# B&R Automation Studio project TD52 (part 82)

#### GridStat.c
```c
/********************************************************************
 * COPYRIGHT -- B&R Industrial Automation GmbH
 ********************************************************************
 * Program: GridStat
 * File: GridStat.c
 * Author: 105055527
 * Last modified by: cadm_kafkama00
 * Created: Mon Sep 05 18:14:57 2016
 * Last modified: Tue Nov 26 15:54:38 2024
 * Model Version: 2.02
 * Description: Detection Algorithm for grid connection.

   HISTORY:
   V1.00  24.07.2020 Keller   created
   V1.01  07.08.2020 Huber  included function block from simulation
   V1.02  29.04.2021 Denk   VectorShift and LVRT function added
   V1.03  31.01.2022 Keller  add input for GCB_On

   V2.00  10.08.2023 Walch  Revision of parametrization, sensitivity and FRT selectivity
   V2.01  22.11.2023 Walch  Include grid observer
   10.01.2024 Walch  Include TP LVRT hold time for weak LVRT blocking
   V2.02  25.11.2024 Walch  Update grid observer for SS mains parallel vs. island plausibility check
 * modified Comment:
 ********************************************************************
 * Implementation of program GridStat
 ********************************************************************
 * Generated with B&R Automation Studio Target for Simulink V6.7.1
 * (ERT based)
 ********************************************************************/

#include "GridStat.h"
#include "GridStat_private.h"

/*  Defines */

/*  Data Types */

/**************************** GLOBAL DATA *************************************/
/*  Definitions */

/*  Declarations  */

/* Forward declaration for local functions */
static real32_T GridStat_mean(const real32_T x[5], struct fGridStat* inst);

/***************************** FILE SCOPE DATA ********************************/

/*************************** FUNCTIONS ****************************************/
int32_T div_nde_s32_floor(int32_T numerator, int32_T denominator, struct fGridStat* inst)
{
  return (((numerator < 0) != (denominator < 0)) && (numerator % denominator !=
           0) ? -1 : 0) + numerator / denominator;
}

/*
 * System initialize for atomic system:
 *    '<S4>/TofLvrtWeakBlk1'
 *    '<S2>/TofMcbFb'
 *    '<S2>/TofReset'
 *    '<S8>/TofAfterFRT'
 *    '<S8>/TofLvrtWeakBlk2'
 */
void GridStat_TofLvrtWeakBlk1_Init(rtDW_TofLvrtWeakBlk1_GridStat *localDW, struct fGridStat* inst)
{
  /* InitializeConditions for DiscreteIntegrator: '<S12>/Discrete-Time Integrator' */
  localDW->DiscreteTimeIntegrator_PrevRese = 2;
  localDW->DiscreteTimeIntegrator_IC_LOADI = 1U;
}

/*
 * Output and update for atomic system:
 *    '<S4>/TofLvrtWeakBlk1'
 *    '<S2>/TofMcbFb'
 *    '<S2>/TofReset'
 *    '<S8>/TofAfterFRT'
 *    '<S8>/TofLvrtWeakBlk2'
 */
void GridStat_TofLvrtWeakBlk1(boolean_T rtu_IN, real32_T rtu_PT,
  rtB_TofLvrtWeakBlk1_GridStat *localB, rtDW_TofLvrtWeakBlk1_GridStat *localDW, struct fGridStat* inst)
{
  real32_T rtb_Switch_l;

  /* Switch: '<S12>/Switch' incorporates:
   *  Constant: '<S12>/Constant1'
   */
  if (rtu_IN) {
    rtb_Switch_l = 0.0F;
  } else {
    rtb_Switch_l = rtu_PT;
  }

  /* End of Switch: '<S12>/Switch' */

  /* DiscreteIntegrator: '<S12>/Discrete-Time Integrator' */
  if (localDW->DiscreteTimeIntegrator_IC_LOADI != 0) {
    localDW->DiscreteTimeIntegrator_DSTATE = rtb_Switch_l;
  }

  if (rtu_IN && (localDW->DiscreteTimeIntegrator_PrevRese <= 0)) {
    localDW->DiscreteTimeIntegrator_DSTATE = rtb_Switch_l;
  }

  /* Logic: '<S12>/Logical Operator1' incorporates:
   *  DiscreteIntegrator: '<S12>/Discrete-Time Integrator'
   *  RelationalOperator: '<S12>/Relational Operator'
   */
  localB->LogicalOperator1 = (localDW->DiscreteTimeIntegrator_DSTATE < rtu_PT);

  /* Update for DiscreteIntegrator: '<S12>/Discrete-Time Integrator' incorporates:
   *  DataTypeConversion: '<S20>/Conversion'
   *  Logic: '<S12>/Logical Operator5'
   */
  localDW->DiscreteTimeIntegrator_IC_LOADI = 0U;
  localDW->DiscreteTimeIntegrator_DSTATE += 0.01F * (real32_T)!rtu_IN;
  localDW->DiscreteTimeIntegrator_PrevRese = (int8_T)rtu_IN;
}

/*
 * System initialize for atomic system:
 *    '<S4>/TpDetNabsProtTrigger'
 *    '<S4>/TpLvrtBlockHold1'
 *    '<S4>/TpLvrtTrigHold1'
 *    '<S4>/TpNabsTrigger'
 *    '<S4>/TpProtTrigger'
 *    '<S8>/TP_PU_trigger'
 *    '<S8>/TpDetVPNTrigger'
 *    '<S8>/TpLvrtBlockHold2'
 *    '<S8>/TpLvrtTrigHold2'
 *    '<S8>/TpNTrigger'
 *    ...
 */
void GridS_TpDetNabsProtTrigger_Init(rtDW_TpDetNabsProtTrigger_GridS *localDW, struct fGridStat* inst)
{
  /* InitializeConditions for UnitDelay: '<S13>/Unit Delay2' */
  localDW->UnitDelay2_DSTATE = true;
}

/*
 * Output and update for atomic system:
 *    '<S4>/TpDetNabsProtTrigger'
 *    '<S4>/TpLvrtBlockHold1'
 *    '<S4>/TpLvrtTrigHold1'
 *    '<S4>/TpNabsTrigger'
 *    '<S4>/TpProtTrigger'
 *    '<S8>/TP_PU_trigger'
 *    '<S8>/TpDetVPNTrigger'
 *    '<S8>/TpLvrtBlockHold2'
 *    '<S8>/TpLvrtTrigHold2'
 *    '<S8>/TpNTrigger'
 *    ...
 */
void GridStat_TpDetNabsProtTrigger(boolean_T rtu_IN, real32_T rtu_PT,
  rtB_TpDetNabsProtTrigger_GridSt *localB, rtDW_TpDetNabsProtTrigger_GridS
  *localDW, struct fGridStat* inst)
{
  real32_T rtb_Switch2;
  real32_T rtb_UkYk1;

  /* Product: '<S24>/delta rise limit' incorporates:
   *  SampleTimeMath: '<S24>/sample time'
   *
   * About '<S24>/sample time':
   *  y = K where K = ( w * Ts )
   */
  rtb_Switch2 = 0.01F;

  /* Outputs for Enabled SubSystem: '<S13>/Enabled Subsystem' incorporates:
   *  EnablePort: '<S22>/Enable'
   */
  /* Logic: '<S13>/Logical Operator3' incorporates:
   *  Logic: '<S13>/Logical Operator2'
   *  UnitDelay: '<S13>/Unit Delay2'
   */
  if ((!rtu_IN) && localDW->UnitDelay2_DSTATE) {
    /* Merge: '<S13>/Merge' incorporates:
     *  Constant: '<S13>/Constant10'
     *  Inport: '<S22>/In1'
     */
    localB->Merge = 0.0F;
  }

  /* End of Logic: '<S13>/Logical Operator3' */
  /* End of Outputs for SubSystem: '<S13>/Enabled Subsystem' */

  /* Outputs for Enabled SubSystem: '<S13>/Enabled Subsystem1' incorporates:
   *  EnablePort: '<S23>/Enable'
   */
  if (rtu_IN) {
    /* Merge: '<S13>/Merge' incorporates:
     *  Inport: '<S23>/In1'
     */
    localB->Merge = rtu_PT;
  }

  /* End of Outputs for SubSystem: '<S13>/Enabled Subsystem1' */

  /* Sum: '<S24>/Difference Inputs1' incorporates:
   *  UnitDelay: '<S24>/Delay Input2'
   */
  rtb_UkYk1 = localB->Merge - localDW->DelayInput2_DSTATE;

  /* Switch: '<S25>/Switch2' incorporates:
   *  RelationalOperator: '<S25>/LowerRelop1'
   */
  if (rtb_UkYk1 <= 0.01F) {
    /* Product: '<S24>/delta fall limit' incorporates:
     *  Constant: '<S13>/Constant9'
     *  SampleTimeMath: '<S24>/sample time'
     *
     * About '<S24>/sample time':
     *  y = K where K = ( w * Ts )
     */
    rtb_Switch2 = -99.99F;

    /* Switch: '<S25>/Switch' incorporates:
     *  RelationalOperator: '<S25>/UpperRelop'
     */
    if (rtb_UkYk1 >= -99.99F) {
      rtb_Switch2 = rtb_UkYk1;
    }

    /* End of Switch: '<S25>/Switch' */
  }

  /* End of Switch: '<S25>/Switch2' */

  /* Sum: '<S24>/Difference Inputs2' incorporates:
   *  UnitDelay: '<S24>/Delay Input2'
   */
  rtb_UkYk1 = rtb_Switch2 + localDW->DelayInput2_DSTATE;

  /* Logic: '<S13>/Logical Operator1' incorporates:
   *  Constant: '<S21>/Constant'
   *  RelationalOperator: '<S13>/Relational Operator1'
   *  RelationalOperator: '<S21>/Compare'
   */
  localB->LogicalOperator1 = ((rtb_UkYk1 > 0.0F) && (rtb_UkYk1 < rtu_PT));

  /* Update for UnitDelay: '<S13>/Unit Delay2' incorporates:
   *  RelationalOperator: '<S13>/Relational Operator3'
   */
  localDW->UnitDelay2_DSTATE = (rtb_UkYk1 >= rtu_PT);

  /* Update for UnitDelay: '<S24>/Delay Input2' */
  localDW->DelayInput2_DSTATE = rtb_UkYk1;
}

/* Function for MATLAB Function: '<S5>/Grid Observer' */
static real32_T GridStat_mean(const real32_T x[5], struct fGridStat* inst)
{
  return ((((x[0] + x[1]) + x[2]) + x[3]) + x[4]) / 5.0F;
}

/* Model step function */
void GridStat_step(RT_MODEL_GridStat *const GridStat_M, struct fGridStat* inst)
{
  struct BlockIO_GridStat *GridStat_B = GridStat_M->blockIO;
  struct D_Work_GridStat *GridStat_DWork = GridStat_M->dwork;
  struct PrevZCSigStates_GridStat *GridStat_PrevZCSigState = GridStat_M->prevZCSigState;
  ExternalOutputs_GridStat *GridStat_Y = (ExternalOutputs_GridStat *)
    GridStat_M->outputs;
  real_T rtb_Switch;
  real_T u0;
  int32_T i;
  int32_T tmp;
  real32_T rtb_Divide4_h;
  real32_T rtb_Product5;
  real32_T rtb_Product6;
  real32_T rtb_Product6_c;
  real32_T rtb_Saturation;
  int16_T rtb_Saturation2;
  int16_T tmp_0;
  boolean_T rtb_AND;
  boolean_T rtb_LogicalOperator3;
  boolean_T rtb_LogicalOperator_b;
  boolean_T rtb_LogicalOperator_i;
  boolean_T rtb_RelationalOperator;
  boolean_T rtb_RelationalOperator3;
  boolean_T rtb_RelationalOperator3_dy;
  boolean_T rtb_RelationalOperator_b;
  boolean_T rtb_Switch6;
  boolean_T rtb_trigger_LVRT_l;
  boolean_T rtb_trigger_N;
  boolean_T rtb_trigger_P;
  boolean_T rtb_trigger_PU;
  boolean_T rtb_trigger_U;

  /* S-Function (bur_bus_in): '<Root>/Bus Input' */
  GridStat_B->BusInput = inst->Para;

  /* S-Function (bur_bus_in): '<Root>/Bus Input2' */
  GridStat_B->BusInput2 = inst->In;

  /* Logic: '<S2>/AND' */
  rtb_AND = (GridStat_B->BusInput2.bGCB_On && GridStat_B->BusInput2.bMCB_On);

  /* Outputs for Atomic SubSystem: '<S2>/TofMcbFb' */
  GridStat_TofLvrtWeakBlk1(rtb_AND, GridStat_B->BusInput.rTi_Tof_MCBfb,
    &GridStat_B->TofMcbFb, &GridStat_DWork->TofMcbFb, inst);

  /* End of Outputs for SubSystem: '<S2>/TofMcbFb' */

  /* Saturate: '<S4>/Saturation5' */
  if (GridStat_B->BusInput.rN_Nom >= 1.0F) {
    rtb_Saturation = GridStat_B->BusInput.rN_Nom;
  } else {
    rtb_Saturation = 1.0F;
  }

  /* End of Saturate: '<S4>/Saturation5' */

  /* RelationalOperator: '<S4>/Relational Operator' incorporates:
   *  Abs: '<S4>/Abs'
   *  Abs: '<S4>/Abs1'
   *  Product: '<S4>/Product4'
   *  Sum: '<S4>/Sum'
   */
  rtb_RelationalOperator = ((real32_T)fabs(GridStat_B->BusInput2.rN_engAct -
    rtb_Saturation) > (real32_T)fabs(rtb_Saturation *
    GridStat_B->BusInput.rThrs_DeltaN_norm));

  /* Outputs for Atomic SubSystem: '<S4>/TpNabsTrigger' */
  /* SignalConversion generated from: '<S4>/Bus Selector2' */
  GridStat_TpDetNabsProtTrigger(rtb_RelationalOperator,
    GridStat_B->BusInput.rTi_Tp_DetectActive, &GridStat_B->TpNabsTrigger,
    &GridStat_DWork->TpNabsTrigger, inst);

  /* End of Outputs for SubSystem: '<S4>/TpNabsTrigger' */

  /* Gain: '<S4>/rpm2omega' */
  rtb_Saturation = 0.104719758F * GridStat_B->BusInput2.rN_engAct;

  /* Outputs for Atomic SubSystem: '<S4>/Speed_filter' */
  /* Logic: '<S11>/Logical Operator' incorporates:
   *  Constant: '<S11>/Constant'
   *  Logic: '<S11>/Logical Operator1'
   *  RelationalOperator: '<S11>/Relational Operator'
   */
  rtb_LogicalOperator_i = (GridStat_B->BusInput2.bReset ||
    (GridStat_B->BusInput.rTi_Filt_speed <= 0.0F));

  /* DiscreteIntegrator: '<S11>/Discrete-Time Integrator' */
  if (GridStat_DWork->DiscreteTimeIntegrator_IC_LOADI != 0) {
    GridStat_DWork->DiscreteTimeIntegrator_DSTATE_j = rtb_Saturation;
  }

  if (rtb_LogicalOperator_i || (GridStat_DWork->DiscreteTimeIntegrator_PrevRese
       != 0)) {
    GridStat_DWork->DiscreteTimeIntegrator_DSTATE_j = rtb_Saturation;
  }

  /* Switch: '<S18>/Switch' incorporates:
   *  Abs: '<S18>/Abs'
   *  RelationalOperator: '<S18>/Relational Operator'
   */
  if (2.22044605E-16F >= (real32_T)fabs(GridStat_B->BusInput.rTi_Filt_speed)) {
    rtb_Product5 = 2.22044605E-16F;
  } else {
    rtb_Product5 = GridStat_B->BusInput.rTi_Filt_speed;
  }

  /* End of Switch: '<S18>/Switch' */

  /* Product: '<S11>/Divide4' incorporates:
   *  DiscreteIntegrator: '<S11>/Discrete-Time Integrator'
   *  Sum: '<S11>/Sum4'
   */
  rtb_Divide4_h = (rtb_Saturation -
                   GridStat_DWork->DiscreteTimeIntegrator_DSTATE_j) /
    rtb_Product5;

  /* Update for DiscreteIntegrator: '<S11>/Discrete-Time Integrator' */
  GridStat_DWork->DiscreteTimeIntegrator_IC_LOADI = 0U;
  GridStat_DWork->DiscreteTimeIntegrator_DSTATE_j += 0.01F * rtb_Divide4_h;
  GridStat_DWork->DiscreteTimeIntegrator_PrevRese = (int8_T)
    rtb_LogicalOperator_i;

  /* End of Outputs for SubSystem: '<S4>/Speed_filter' */

  /* Gain: '<S4>/W2kW' */
  rtb_Product6 = 1000.0F * GridStat_B->BusInput.rP_Nom;

  /* Outputs for Atomic SubSystem: '<S4>/Speed_filter' */
  /* Switch: '<S11>/Switch1' incorporates:
   *  Constant: '<S11>/Constant'
   */
  if (rtb_LogicalOperator_i) {
    rtb_Divide4_h = 0.0F;
  }

  /* End of Switch: '<S11>/Switch1' */
  /* End of Outputs for SubSystem: '<S4>/Speed_filter' */

  /* Saturate: '<S4>/Saturation' */
  if (rtb_Product6 < 1.0F) {
    rtb_Product6 = 1.0F;
  }

  /* End of Saturate: '<S4>/Saturation' */

  /* Product: '<S4>/Product2' incorporates:
   *  Product: '<S4>/Product1'
   */
  rtb_Saturation = rtb_Saturation * rtb_Divide4_h *
    GridStat_B->BusInput.rJ_Engine / rtb_Product6;

  /* RelationalOperator: '<S4>/Relational Operator2' */
  rtb_LogicalOperator_i = (rtb_Saturation >
    GridStat_B->BusInput.rProt_Norm_limit);

  /* Outputs for Atomic SubSystem: '<S4>/TpProtTrigger' */
  /* SignalConversion generated from: '<S4>/Bus Selector2' */
  GridStat_TpDetNabsProtTrigger(rtb_LogicalOperator_i,
    GridStat_B->BusInput.rTi_Tp_DetectActive, &GridStat_B->TpProtTrigger,
    &GridStat_DWork->TpProtTrigger, inst);

  /* End of Outputs for SubSystem: '<S4>/TpProtTrigger' */

  /* RelationalOperator: '<S4>/Relational Operator3' */
  rtb_RelationalOperator3 = (GridStat_B->BusInput2.rU_norm <=
    GridStat_B->BusInput.rThrs_LVRT_norm);

  /* Saturate: '<S4>/Saturation1' */
  if (GridStat_B->BusInput.rTi_sampleRate >= 0.001F) {
    /* Saturate: '<S8>/Saturation' incorporates:
     *  Saturate: '<S8>/Saturation1'
     */
    rtb_Divide4_h = GridStat_B->BusInput.rTi_sampleRate;
  } else {
    /* Saturate: '<S8>/Saturation' incorporates:
     *  Saturate: '<S8>/Saturation1'
     */
    rtb_Divide4_h = 0.001F;
  }

  /* Saturate: '<S4>/Saturation4' incorporates:
   *  DataTypeConversion: '<S4>/Cast1'
   */
  if (GridStat_B->BusInput.iSamples_Tp_LVRT_hold > 10000.0F) {
    rtb_Product5 = 10000.0F;
  } else if (GridStat_B->BusInput.iSamples_Tp_LVRT_hold < 1.0F) {
    rtb_Product5 = 1.0F;
  } else {
    rtb_Product5 = GridStat_B->BusInput.iSamples_Tp_LVRT_hold;
  }

  /* End of Saturate: '<S4>/Saturation4' */

  /* Product: '<S4>/Product6' incorporates:
   *  Saturate: '<S4>/Saturation1'
   */
  rtb_Product6 = rtb_Divide4_h * rtb_Product5;

  /* Outputs for Atomic SubSystem: '<S4>/TpLvrtBlockHold1' */
  /* Logic: '<S4>/Logical Operator2' */
  GridStat_TpDetNabsProtTrigger((rtb_RelationalOperator3 ||
    GridStat_B->BusInput2.bLVRT), rtb_Product6, &GridStat_B->TpLvrtBlockHold1,
    &GridStat_DWork->TpLvrtBlockHold1, inst);

  /* End of Outputs for SubSystem: '<S4>/TpLvrtBlockHold1' */

  /* Saturate: '<S4>/Saturation2' incorporates:
   *  Constant: '<S4>/Constant1'
   *  DataTypeConversion: '<S4>/Cast'
   *  Sum: '<S4>/Sum3'
   */
  if (10.0F - (real32_T)GridStat_B->BusInput.iSensitivity_WeakBlocking > 10.0F)
  {
    rtb_Product5 = 10.0F;
  } else if (10.0F - (real32_T)GridStat_B->BusInput.iSensitivity_WeakBlocking <
             1.0F) {
    rtb_Product5 = 1.0F;
  } else {
    rtb_Product5 = 10.0F - (real32_T)
      GridStat_B->BusInput.iSensitivity_WeakBlocking;
  }

  /* End of Saturate: '<S4>/Saturation2' */

  /* Outputs for Atomic SubSystem: '<S4>/TofLvrtWeakBlk1' */
  /* Product: '<S4>/Product7' incorporates:
   *  Saturate: '<S4>/Saturation1'
   */
  GridStat_TofLvrtWeakBlk1(rtb_RelationalOperator3, rtb_Product5 * rtb_Divide4_h,
    &GridStat_B->TofLvrtWeakBlk1, &GridStat_DWork->TofLvrtWeakBlk1, inst);

  /* End of Outputs for SubSystem: '<S4>/TofLvrtWeakBlk1' */

  /* Outputs for Atomic SubSystem: '<S4>/TpLvrtTrigHold1' */
  GridStat_TpDetNabsProtTrigger(GridStat_B->BusInput2.bLVRT, rtb_Product6,
    &GridStat_B->TpLvrtTrigHold1, &GridStat_DWork->TpLvrtTrigHold1, inst);

  /* End of Outputs for SubSystem: '<S4>/TpLvrtTrigHold1' */

  /* Switch: '<S4>/Switch1' incorporates:
   *  Constant: '<S4>/Constant'
   *  Logic: '<S4>/Logical Operator1'
   *  Logic: '<S4>/Logical Operator11'
   *  Logic: '<S4>/Logical Operator3'
   *  Logic: '<S4>/NOT2'
   *  Switch: '<S4>/Switch5'
   */
  if (rtb_RelationalOperator && (GridStat_B->BusInput.bN_BypassFRTBlocking &&
       GridStat_B->BusInput.bN_BypassFRTBlocking_speedAbs)) {
    rtb_RelationalOperator3 = false;
  } else if ((!GridStat_B->BusInput.bWeakFRTBlocking) ||
             (!GridStat_B->BusInput.bWeakFRTBlocking_speedAbs)) {
    /* Switch: '<S4>/Switch5' */
    rtb_RelationalOperator3 = GridStat_B->TpLvrtBlockHold1.LogicalOperator1;
  } else {
    /* Switch: '<S4>/Switch5' incorporates:
     *  Logic: '<S4>/Logical Operator9'
     */
    rtb_RelationalOperator3 = (GridStat_B->TofLvrtWeakBlk1.LogicalOperator1 &&
      GridStat_B->TpLvrtTrigHold1.LogicalOperator1);
  }

  /* End of Switch: '<S4>/Switch1' */

  /* Logic: '<S4>/NOT' */
  rtb_Switch6 = !rtb_RelationalOperator3;

  /* Switch: '<S4>/Switch4' incorporates:
   *  Saturate: '<S4>/Saturation1'
   */
  if (rtb_Switch6) {
    rtb_Product6 = GridStat_B->BusInput.rTi_Tp_DetectActive;
  } else {
    rtb_Product6 = rtb_Divide4_h;
  }

  /* End of Switch: '<S4>/Switch4' */

  /* Outputs for Atomic SubSystem: '<S4>/TpDetNabsProtTrigger' */
  /* Logic: '<S4>/Logical Operator4' incorporates:
   *  Logic: '<S4>/Logical Operator'
   */
  GridStat_TpDetNabsProtTrigger(((GridStat_B->TpNabsTrigger.LogicalOperator1 ||
    GridStat_B->TpProtTrigger.LogicalOperator1) && rtb_Switch6), rtb_Product6,
    &GridStat_B->TpDetNabsProtTrigger, &GridStat_DWork->TpDetNabsProtTrigger, inst);

  /* End of Outputs for SubSystem: '<S4>/TpDetNabsProtTrigger' */

  /* Saturate: '<S8>/Saturation2' */
  if (GridStat_B->BusInput.iSamples_derivative_PU > 10) {
    rtb_Saturation2 = 10;
  } else if (GridStat_B->BusInput.iSamples_derivative_PU < 1) {
    rtb_Saturation2 = 1;
  } else {
    rtb_Saturation2 = GridStat_B->BusInput.iSamples_derivative_PU;
  }

  /* End of Saturate: '<S8>/Saturation2' */

  /* Product: '<S8>/Product' */
  rtb_Product6 = (real32_T)rtb_Saturation2 * rtb_Divide4_h;

  /* RelationalOperator: '<S8>/Relational Operator3' */
  rtb_RelationalOperator3_dy = (GridStat_B->BusInput2.rU_norm <=
    GridStat_B->BusInput.rThrs_LVRT_norm);

  /* Saturate: '<S8>/Saturation7' incorporates:
   *  Constant: '<S8>/Constant1'
   *  DataTypeConversion: '<S8>/Cast'
   *  Sum: '<S8>/Sum3'
   */
  if (10.0F - (real32_T)GridStat_B->BusInput.iSensitivity_WeakBlocking > 10.0F)
  {
    rtb_Product5 = 10.0F;
  } else if (10.0F - (real32_T)GridStat_B->BusInput.iSensitivity_WeakBlocking <
             1.0F) {
    rtb_Product5 = 1.0F;
  } else {
    rtb_Product5 = 10.0F - (real32_T)
      GridStat_B->BusInput.iSensitivity_WeakBlocking;
  }

  /* End of Saturate: '<S8>/Saturation7' */

  /* Outputs for Atomic SubSystem: '<S8>/TofLvrtWeakBlk2' */
  /* Product: '<S8>/Product7' */
  GridStat_TofLvrtWeakBlk1(rtb_RelationalOperator3_dy, rtb_Product5 *
    rtb_Divide4_h, &GridStat_B->TofLvrtWeakBlk2,
    &GridStat_DWork->TofLvrtWeakBlk2, inst);

  /* End of Outputs for SubSystem: '<S8>/TofLvrtWeakBlk2' */

  /* Saturate: '<S8>/Saturation4' */
  if (GridStat_B->BusInput.iSamples_Tp_LVRT_hold > 10000) {
    tmp_0 = 10000;
  } else if (GridStat_B->BusInput.iSamples_Tp_LVRT_hold < 1) {
    tmp_0 = 1;
  } else {
    tmp_0 = GridStat_B->BusInput.iSamples_Tp_LVRT_hold;
  }

  /* End of Saturate: '<S8>/Saturation4' */

  /* Product: '<S8>/Product6' */
  rtb_Product6_c = rtb_Divide4_h * (real32_T)tmp_0;

  /* Outputs for Atomic SubSystem: '<S8>/TpLvrtTrigHold2' */
  GridStat_TpDetNabsProtTrigger(GridStat_B->BusInput2.bLVRT, rtb_Product6_c,
    &GridStat_B->TpLvrtTrigHold2, &GridStat_DWork->TpLvrtTrigHold2, inst);

  /* End of Outputs for SubSystem: '<S8>/TpLvrtTrigHold2' */

  /* Logic: '<S8>/Logical Operator9' */
  rtb_trigger_LVRT_l = (GridStat_B->TofLvrtWeakBlk2.LogicalOperator1 &&
                        GridStat_B->TpLvrtTrigHold2.LogicalOperator1);

  /* Saturate: '<S8>/Saturation6' */
  if (GridStat_B->BusInput.iSamples_Tof_U_norm_FRTBlock > 1000) {
    tmp_0 = 1000;
  } else if (GridStat_B->BusInput.iSamples_Tof_U_norm_FRTBlock < 1) {
    tmp_0 = 1;
  } else {
    tmp_0 = GridStat_B->BusInput.iSamples_Tof_U_norm_FRTBlock;
  }

  /* End of Saturate: '<S8>/Saturation6' */

  /* Outputs for Atomic SubSystem: '<S8>/TofAfterFRT' */
  /* Product: '<S8>/Product8' */
  GridStat_TofLvrtWeakBlk1(rtb_trigger_LVRT_l, (real32_T)tmp_0 * rtb_Divide4_h,
    &GridStat_B->TofAfterFRT, &GridStat_DWork->TofAfterFRT, inst);

  /* End of Outputs for SubSystem: '<S8>/TofAfterFRT' */

  /* Switch: '<S8>/Switch7' incorporates:
   *  Logic: '<S8>/NOT3'
   */
  if (!GridStat_B->TofAfterFRT.LogicalOperator1) {
    rtb_Product5 = GridStat_B->BusInput.rThrs_U_norm;
  } else {
    rtb_Product5 = GridStat_B->BusInput.rThrs_U_norm_FRTBlock;
  }

  /* End of Switch: '<S8>/Switch7' */

  /* RelationalOperator: '<S8>/Relational Operator' incorporates:
   *  Abs: '<S8>/Abs'
   *  Product: '<S8>/Product1'
   *  S-Function (sfix_udelay): '<S8>/Tapped Delay'
   *  Selector: '<S8>/Selector'
   *  Sum: '<S8>/Sum'
   */
  rtb_trigger_U = ((real32_T)fabs(GridStat_DWork->TappedDelay_X[rtb_Saturation2
    - 1] - GridStat_B->BusInput2.rU_norm) / rtb_Product6 >= rtb_Product5);

  /* Saturate: '<S8>/Saturation3' */
  if (GridStat_B->BusInput.iSamples_Tp_detect_VPN > 1000) {
    tmp_0 = 1000;
  } else if (GridStat_B->BusInput.iSamples_Tp_detect_VPN < 1) {
    tmp_0 = 1;
  } else {
    tmp_0 = GridStat_B->BusInput.iSamples_Tp_detect_VPN;
  }

  /* End of Saturate: '<S8>/Saturation3' */

  /* Product: '<S8>/Product5' */
  rtb_Product5 = (real32_T)tmp_0 * rtb_Divide4_h;

  /* Outputs for Atomic SubSystem: '<S8>/TpUTrigger' */
  GridStat_TpDetNabsProtTrigger(rtb_trigger_U, rtb_Product5,
    &GridStat_B->TpUTrigger, &GridStat_DWork->TpUTrigger, inst);

  /* End of Outputs for SubSystem: '<S8>/TpUTrigger' */

  /* RelationalOperator: '<S8>/Relational Operator1' incorporates:
   *  Abs: '<S8>/Abs1'
   *  Product: '<S8>/Product2'
   *  S-Function (sfix_udelay): '<S8>/Tapped Delay1'
   *  Selector: '<S8>/Selector'
   *  Selector: '<S8>/Selector1'
   *  Sum: '<S8>/Sum1'
   */
  rtb_trigger_P = ((real32_T)fabs(GridStat_DWork->TappedDelay1_X[rtb_Saturation2
    - 1] - GridStat_B->BusInput2.rP_norm) / rtb_Product6 >=
                   GridStat_B->BusInput.rThrs_P_norm);

  /* Outputs for Atomic SubSystem: '<S8>/TpPTrigger' */
  GridStat_TpDetNabsProtTrigger(rtb_trigger_P, rtb_Product5,
    &GridStat_B->TpPTrigger, &GridStat_DWork->TpPTrigger, inst);

  /* End of Outputs for SubSystem: '<S8>/TpPTrigger' */

  /* Switch: '<S8>/Switch1' incorporates:
   *  Logic: '<S8>/Logical Operator5'
   *  Logic: '<S8>/Logical Operator6'
   *  Switch: '<S8>/Switch'
   */
  if (GridStat_B->BusInput.bLimitedTriggerTime) {
    rtb_RelationalOperator_b = GridStat_B->TpUTrigger.LogicalOperator1;
    rtb_LogicalOperator3 = GridStat_B->TpPTrigger.LogicalOperator1;
  } else {
    rtb_RelationalOperator_b = (GridStat_B->TpUTrigger.LogicalOperator1 ||
      rtb_trigger_U);
    rtb_LogicalOperator3 = (GridStat_B->TpPTrigger.LogicalOperator1 ||
      rtb_trigger_P);
  }

  /* End of Switch: '<S8>/Switch1' */

  /* Logic: '<S8>/Logical Operator' */
  rtb_trigger_PU = (rtb_RelationalOperator_b && rtb_LogicalOperator3);

  /* Outputs for Atomic SubSystem: '<S8>/TP_PU_trigger' */
  GridStat_TpDetNabsProtTrigger(rtb_trigger_PU, rtb_Product5,
    &GridStat_B->TP_PU_trigger, &GridStat_DWork->TP_PU_trigger, inst);

  /* End of Outputs for SubSystem: '<S8>/TP_PU_trigger' */

  /* Saturate: '<S8>/Saturation5' */
  if (GridStat_B->BusInput.iSamples_derivative_N > 10) {
    rtb_Saturation2 = 10;
  } else if (GridStat_B->BusInput.iSamples_derivative_N < 1) {
    rtb_Saturation2 = 1;
  } else {
    rtb_Saturation2 = GridStat_B->BusInput.iSamples_derivative_N;
  }

  /* End of Saturate: '<S8>/Saturation5' */

  /* RelationalOperator: '<S8>/Relational Operator2' incorporates:
   *  Abs: '<S8>/Abs2'
   *  Product: '<S8>/Product3'
   *  Product: '<S8>/Product4'
   *  S-Function (sfix_udelay): '<S8>/Tapped Delay2'
   *  Selector: '<S8>/Selector2'
   *  Sum: '<S8>/Sum2'
   */
  rtb_trigger_N = (GridStat_B->BusInput.rThrs_N_eng <= 1.0F / (rtb_Divide4_h *
    (real32_T)rtb_Saturation2) * (real32_T)fabs(GridStat_DWork->
    TappedDelay2_X[rtb_Saturation2 - 1] - GridStat_B->BusInput2.rN_engAct));

  /* Outputs for Atomic SubSystem: '<S8>/TpNTrigger' */
  GridStat_TpDetNabsProtTrigger(rtb_trigger_N, rtb_Product5,
    &GridStat_B->TpNTrigger, &GridStat_DWork->TpNTrigger, inst);

  /* End of Outputs for SubSystem: '<S8>/TpNTrigger' */

  /* Outputs for Atomic SubSystem: '<S8>/TpLvrtBlockHold2' */
  /* Logic: '<S8>/Logical Operator2' */
  GridStat_TpDetNabsProtTrigger((rtb_RelationalOperator3_dy ||
    GridStat_B->BusInput2.bLVRT), rtb_Product6_c, &GridStat_B->TpLvrtBlockHold2,
    &GridStat_DWork->TpLvrtBlockHold2, inst);

  /* End of Outputs for SubSystem: '<S8>/TpLvrtBlockHold2' */

  /* Switch: '<S8>/Switch6' incorporates:
   *  Constant: '<S8>/Constant'
   *  Logic: '<S8>/Logical Operator10'
   *  Logic: '<S8>/Logical Operator11'
   *  Logic: '<S8>/Logical Operator12'
   *  Logic: '<S8>/NOT2'
   *  Switch: '<S8>/Switch5'
   */
  if (rtb_RelationalOperator && (GridStat_B->BusInput.bN_BypassFRTBlocking &&
       GridStat_B->BusInput.bN_BypassFRTBlocking_VPN)) {
    rtb_Switch6 = false;
  } else if ((!GridStat_B->BusInput.bWeakFRTBlocking) ||
             (!GridStat_B->BusInput.bWeakFRTBlocking_VPN)) {
    /* Switch: '<S8>/Switch5' */
    rtb_Switch6 = GridStat_B->TpLvrtBlockHold2.LogicalOperator1;
  } else {
    rtb_Switch6 = rtb_trigger_LVRT_l;
  }

  /* End of Switch: '<S8>/Switch6' */

  /* Logic: '<S8>/NOT' */
  rtb_trigger_LVRT_l = !rtb_Switch6;

  /* Switch: '<S8>/Switch2' incorporates:
   *  Logic: '<S8>/Logical Operator7'
   */
  if (GridStat_B->BusInput.bLimitedTriggerTime) {
    rtb_RelationalOperator_b = GridStat_B->TP_PU_trigger.LogicalOperator1;
  } else {
    rtb_RelationalOperator_b = (GridStat_B->TP_PU_trigger.LogicalOperator1 ||
      rtb_trigger_PU);
  }

  /* End of Switch: '<S8>/Switch2' */

  /* Switch: '<S8>/Switch3' incorporates:
   *  Logic: '<S8>/Logical Operator8'
   *  Logic: '<S8>/NOT1'
   */
  if (!GridStat_B->BusInput.bLimitedTriggerTime) {
    rtb_LogicalOperator3 = (rtb_trigger_N ||
      GridStat_B->TpNTrigger.LogicalOperator1);
  } else {
    rtb_LogicalOperator3 = GridStat_B->TpNTrigger.LogicalOperator1;
  }

  /* End of Switch: '<S8>/Switch3' */

  /* Switch: '<S8>/Switch4' */
  if (rtb_trigger_LVRT_l) {
    rtb_Divide4_h = GridStat_B->BusInput.rTi_Tp_DetectActive;
  }

  /* End of Switch: '<S8>/Switch4' */

  /* Outputs for Atomic SubSystem: '<S8>/TpDetVPNTrigger' */
  /* Logic: '<S8>/Logical Operator4' incorporates:
   *  Logic: '<S8>/Logical Operator1'
   *  Logic: '<S8>/Logical Operator3'
   */
  GridStat_TpDetNabsProtTrigger((((rtb_RelationalOperator_b &&
    rtb_LogicalOperator3) || GridStat_B->BusInput2.bVectorShift) &&
    rtb_trigger_LVRT_l), rtb_Divide4_h, &GridStat_B->TpDetVPNTrigger,
    &GridStat_DWork->TpDetVPNTrigger, inst);

  /* End of Outputs for SubSystem: '<S8>/TpDetVPNTrigger' */

  /* MATLAB Function: '<S5>/Grid Observer' */
  /* MATLAB Function 'detection + correction: transition to Island/Smooth Detection/Grid Observer': '<S52>:1' */
  /* '<S52>:1:2' */
  tmp = 10 - GridStat_B->BusInput.iSensitivity_SmoothDetection;
  if (10 - GridStat_B->BusInput.iSensitivity_SmoothDetection > 32767) {
    tmp = 32767;
  }

  if ((!GridStat_DWork->U_past_not_empty) || GridStat_B->BusInput2.bReset) {
    GridStat_DWork->ctr_U = 0;
    for (i = 0; i < 1000; i++) {
      GridStat_DWork->U_past[i] = GridStat_B->BusInput2.rU_norm;
    }

    GridStat_DWork->U_past_not_empty = true;
  }

  i = GridStat_DWork->ctr_U + 1;
  if (GridStat_DWork->ctr_U + 1 > 32767) {
    i = 32767;
  }

  GridStat_DWork->U_past[i - 1] = GridStat_B->BusInput2.rU_norm;
  rtb_Divide4_h = 0.0F;
  for (rtb_Saturation2 = 0; rtb_Saturation2 < 1000; rtb_Saturation2++) {
    i = GridStat_DWork->ctr_U - rtb_Saturation2;
    if (i < -32768) {
      i = -32768;
    }

    i = (int16_T)((int16_T)i - (int16_T)((int16_T)div_nde_s32_floor((int16_T)i,
      1000, inst) * 1000)) + 1;
    if (i > 32767) {
      i = 32767;
    }

    rtb_Divide4_h += GridStat_DWork->U_past[i - 1];
  }

  rtb_Divide4_h /= 1000.0F;
  i = GridStat_DWork->ctr_U + 1;
  if (GridStat_DWork->ctr_U + 1 > 32767) {
    i = 32767;
  }

  GridStat_DWork->ctr_U = (int16_T)i;
  if (GridStat_DWork->ctr_U >= 1000) {
    GridStat_DWork->ctr_U = 0;
  }

  if ((!GridStat_DWork->err_past_not_empty) || GridStat_B->BusInput2.bReset) {
    GridStat_DWork->ctr_err = 0;
    GridStat_DWork->ctr_acterr = 0;
    GridStat_DWork->ctr_release = 0;
    for (i = 0; i < 1000; i++) {
      GridStat_DWork->err_past[i] = 0.0F;
    }

    GridStat_DWork->err_past_not_empty = true;
    GridStat_DWork->err_min = 1.0E+6F;
    GridStat_DWork->err_act = 0.0F;
    GridStat_DWork->err_max = 0.0F;
    GridStat_DWork->flag_window = true;
    for (i = 0; i < 5; i++) {
      GridStat_DWork->err_act_temp[i] = 0.0F;
    }
  }

  i = GridStat_DWork->ctr_err + 1;
  if (GridStat_DWork->ctr_err + 1 > 32767) {
    i = 32767;
  }

  if (1.0F >= GridStat_B->BusInput.rN_Nom) {
    rtb_Product5 = 1.0F;
  } else {
    rtb_Product5 = GridStat_B->BusInput.rN_Nom;
  }

  GridStat_DWork->err_past[i - 1] = (real32_T)fabs
    (GridStat_B->BusInput2.rN_engAct / rtb_Product5 - 1.0F);
  rtb_Product6 = GridStat_DWork->err_past[0];
  for (i = 0; i < 999; i++) {
    rtb_Product6 += GridStat_DWork->err_past[i + 1];
  }

  rtb_trigger_LVRT_l = true;
  if (GridStat_DWork->ctr_release < 6000) {
    i = GridStat_DWork->ctr_release + 1;
    if (GridStat_DWork->ctr_release + 1 > 32767) {
      i = 32767;
    }

    GridStat_DWork->ctr_release = (int16_T)i;
    rtb_trigger_LVRT_l = false;
  }

  if (GridStat_DWork->flag_window && rtb_trigger_LVRT_l) {
    i = GridStat_DWork->ctr_acterr + 1;
    if (GridStat_DWork->ctr_acterr + 1 > 32767) {
      i = 32767;
    }

    GridStat_DWork->err_act_temp[i - 1] = rtb_Product6 / 1000.0F;
    i = GridStat_DWork->ctr_acterr + 1;
    if (GridStat_DWork->ctr_acterr + 1 > 32767) {
      i = 32767;
    }

    GridStat_DWork->ctr_acterr = (int16_T)i;
    GridStat_DWork->flag_window = false;
  }

  rtb_Product6 = GridStat_DWork->err_act_temp[0];
  rtb_Product6_c = GridStat_mean(GridStat_DWork->err_act_temp, inst);
  rtb_Product5 = GridStat_DWork->err_act_temp[0];
  if (GridStat_DWork->err_act_temp[0] < GridStat_DWork->err_act_temp[1]) {
    rtb_Product6 = GridStat_DWork->err_act_temp[1];
  }

  if (GridStat_DWork->err_act_temp[0] > GridStat_DWork->err_act_temp[1]) {
    rtb_Product5 = GridStat_DWork->err_act_temp[1];
  }

  if (rtb_Product6 < GridStat_DWork->err_act_temp[2]) {
    rtb_Product6 = GridStat_DWork->err_act_temp[2];
  }

  if (rtb_Product5 > GridStat_DWork->err_act_temp[2]) {
    rtb_Product5 = GridStat_DWork->err_act_temp[2];
  }

  if (rtb_Product6 < GridStat_DWork->err_act_temp[3]) {
    rtb_Product6 = GridStat_DWork->err_act_temp[3];
  }

  if (rtb_Product5 > GridStat_DWork->err_act_temp[3]) {
    rtb_Product5 = GridStat_DWork->err_act_temp[3];
  }

  if (rtb_Product6 < GridStat_DWork->err_act_temp[4]) {
    rtb_Product6 = GridStat_DWork->err_act_temp[4];
  }

  if (rtb_Product5 > GridStat_DWork->err_act_temp[4]) {
    rtb_Product5 = GridStat_DWork->err_act_temp[4];
  }

  if (((real32_T)fabs(rtb_Product6 - rtb_Product6_c) < rtb_Product6_c) &&
      ((real32_T)fabs(rtb_Product6_c - rtb_Product5) < rtb_Product6_c)) {
    GridStat_DWork->err_act = GridStat_mean(GridStat_DWork->err_act_temp, inst);
  }

  if ((GridStat_DWork->err_act < GridStat_DWork->err_min) &&
      (GridStat_DWork->err_act > 1.0E-8F)) {
    GridStat_DWork->err_min = GridStat_DWork->err_act;
  }

  if (GridStat_DWork->err_act > GridStat_DWork->err_max) {
    GridStat_DWork->err_max = GridStat_DWork->err_act;
  }

  if (GridStat_DWork->ctr_acterr > 4) {
    GridStat_DWork->ctr_acterr = 0;
  }

  i = GridStat_DWork->ctr_err + 1;
  if (GridStat_DWork->ctr_err + 1 > 32767) {
    i = 32767;
  }

  GridStat_DWork->ctr_err = (int16_T)i;
  if (GridStat_DWork->ctr_err >= 1000) {
    GridStat_DWork->ctr_err = 0;
    GridStat_DWork->flag_window = true;
  }

  if ((!GridStat_DWork->err_past_Q_not_empty) || GridStat_B->BusInput2.bReset) {
    GridStat_DWork->ctr_err_Q = 0;
    GridStat_DWork->ctr_acterr_Q = 0;
    GridStat_DWork->ctr_release_Q = 0;
    for (i = 0; i < 1000; i++) {
      GridStat_DWork->err_past_Q[i] = 0.0F;
    }

    GridStat_DWork->err_past_Q_not_empty = true;
    GridStat_DWork->err_min_Q = 1.0E+6F;
    GridStat_DWork->err_act_Q = 0.0F;
    GridStat_DWork->err_max_Q = 0.0F;
    GridStat_DWork->flag_window_Q = true;
    for (i = 0; i < 5; i++) {
      GridStat_DWork->err_act_temp_Q[i] = 0.0F;
    }
  }

  i = GridStat_DWork->ctr_err_Q + 1;
  if (GridStat_DWork->ctr_err_Q + 1 > 32767) {
    i = 32767;
  }

  GridStat_DWork->err_past_Q[i - 1] = (real32_T)fabs
    (GridStat_B->BusInput2.rU_norm - rtb_Divide4_h);
  rtb_Divide4_h = GridStat_DWork->err_past_Q[0];
  for (i = 0; i < 999; i++) {
    rtb_Divide4_h += GridStat_DWork->err_past_Q[i + 1];
  }

  rtb_trigger_LVRT_l = true;
  if (GridStat_DWork->ctr_release_Q < 6000) {
    i = GridStat_DWork->ctr_release_Q + 1;
    if (GridStat_DWork->ctr_release_Q + 1 > 32767) {
      i = 32767;
    }

    GridStat_DWork->ctr_release_Q = (int16_T)i;
    rtb_trigger_LVRT_l = false;
  }

  if (GridStat_DWork->flag_window_Q && rtb_trigger_LVRT_l) {
    i = GridStat_DWork->ctr_acterr_Q + 1;
    if (GridStat_DWork->ctr_acterr_Q + 1 > 32767) {
      i = 32767;
    }

    GridStat_DWork->err_act_temp_Q[i - 1] = rtb_Divide4_h / 1000.0F;
    i = GridStat_DWork->ctr_acterr_Q + 1;
    if (GridStat_DWork->ctr_acterr_Q + 1 > 32767) {
      i = 32767;
    }

    GridStat_DWork->ctr_acterr_Q = (int16_T)i;
    GridStat_DWork->flag_window_Q = false;
  }

  rtb_Divide4_h = GridStat_DWork->err_act_temp_Q[0];
  rtb_Product6 = GridStat_mean(GridStat_DWork->err_act_temp_Q, inst);
  rtb_Product6_c = GridStat_DWork->err_act_temp_Q[0];
  if (GridStat_DWork->err_act_temp_Q[0] < GridStat_DWork->err_act_temp_Q[1]) {
    rtb_Divide4_h = GridStat_DWork->err_act_temp_Q[1];
  }

  if (GridStat_DWork->err_act_temp_Q[0] > GridStat_DWork->err_act_temp_Q[1]) {
    rtb_Product6_c = GridStat_DWork->err_act_temp_Q[1];
  }

  if (rtb_Divide4_h < GridStat_DWork->err_act_temp_Q[2]) {
    rtb_Divide4_h = GridStat_DWork->err_act_temp_Q[2];
  }

  if (rtb_Product6_c > GridStat_DWork->err_act_temp_Q[2]) {
    rtb_Product6_c = GridStat_DWork->err_act_temp_Q[2];
  }

  if (rtb_Divide4_h < GridStat_DWork->err_act_temp_Q[3]) {
    rtb_Divide4_h = GridStat_DWork->err_act_temp_Q[3];
  }

  if (rtb_Product6_c > GridStat_DWork->err_act_temp_Q[3]) {
    rtb_Product6_c = GridStat_DWork->err_act_temp_Q[3];
  }

  if (rtb_Divide4_h < GridStat_DWork->err_act_temp_Q[4]) {
    rtb_Divide4_h = GridStat_DWork->err_act_temp_Q[4];
  }

  if (rtb_Product6_c > GridStat_DWork->err_act_temp_Q[4]) {
    rtb_Product6_c = GridStat_DWork->err_act_temp_Q[4];
  }

  if (((real32_T)fabs(rtb_Divide4_h - rtb_Product6) < rtb_Product6) &&
      ((real32_T)fabs(rtb_Product6 - rtb_Product6_c) < rtb_Product6)) {
    GridStat_DWork->err_act_Q = GridStat_mean(GridStat_DWork->err_act_temp_Q, inst);
  }

  if ((GridStat_DWork->err_act_Q < GridStat_DWork->err_min_Q) &&
      (GridStat_DWork->err_act_Q > 1.0E-8F)) {
    GridStat_DWork->err_min_Q = GridStat_DWork->err_act_Q;
  }

  if (GridStat_DWork->err_act_Q > GridStat_DWork->err_max_Q) {
    GridStat_DWork->err_max_Q = GridStat_DWork->err_act_Q;
  }

  if (GridStat_DWork->ctr_acterr_Q > 4) {
    GridStat_DWork->ctr_acterr_Q = 0;
  }

  i = GridStat_DWork->ctr_err_Q + 1;
  if (GridStat_DWork->ctr_err_Q + 1 > 32767) {
    i = 32767;
  }

  GridStat_DWork->ctr_err_Q = (int16_T)i;
  if (GridStat_DWork->ctr_err_Q >= 1000) {
    GridStat_DWork->ctr_err_Q = 0;
    GridStat_DWork->flag_window_Q = true;
  }

  rtb_RelationalOperator_b = false;
  rtb_Divide4_h = (real32_T)(int16_T)tmp / 2.0F;
  if ((int16_T)tmp == 0) {
    rtb_Divide4_h = 0.25F;
  }

  if (1.0E-8F >= GridStat_DWork->err_min) {
    rtb_Product5 = 1.0E-8F;
  } else {
    rtb_Product5 = GridStat_DWork->err_min;
  }

  if (GridStat_DWork->err_act / rtb_Product5 > rtb_Divide4_h * 15.0F) {
    rtb_RelationalOperator_b = true;
  } else {
    if (1.0E-8F >= GridStat_DWork->err_min_Q) {
      rtb_Product5 = 1.0E-8F;
    } else {
      rtb_Product5 = GridStat_DWork->err_min_Q;
    }

    if (GridStat_DWork->err_act_Q / rtb_Product5 > rtb_Divide4_h * 3.5F) {
      rtb_RelationalOperator_b = true;
    }
  }

  /* MultiPortSwitch: '<S2>/Multiport Switch' incorporates:
   *  Logic: '<S2>/Logical Operator'
   *  Logic: '<S2>/Logical Operator1'
   */
  /* '<S52>:1:2' */
  switch (GridStat_B->BusInput.iDetectMode) {
   case 1:
    rtb_trigger_LVRT_l = GridStat_B->TpDetNabsProtTrigger.LogicalOperator1;
    break;

   case 2:
    rtb_trigger_LVRT_l = GridStat_B->TpDetVPNTrigger.LogicalOperator1;
    break;

   default:
    rtb_trigger_LVRT_l = (GridStat_B->TpDetNabsProtTrigger.LogicalOperator1 ||
                          GridStat_B->TpDetVPNTrigger.LogicalOperator1 ||
                          (GridStat_B->BusInput.bEnable_SmoothDetection &&
      rtb_RelationalOperator_b));
    break;
  }

  /* End of MultiPortSwitch: '<S2>/Multiport Switch' */

  /* Logic: '<S2>/Logical Operator3' incorporates:
   *  Logic: '<S2>/Logical Operator5'
   */
  rtb_LogicalOperator3 = ((rtb_AND || GridStat_B->TofMcbFb.LogicalOperator1) &&
    GridStat_B->BusInput.bEnable && rtb_trigger_LVRT_l);

  /* Outputs for Atomic SubSystem: '<S2>/TofReset' */
  GridStat_TofLvrtWeakBlk1(rtb_LogicalOperator3,
    GridStat_B->BusInput.rTi_Filt_factorNoffsetCorr, &GridStat_B->TofReset,
    &GridStat_DWork->TofReset, inst);

  /* End of Outputs for SubSystem: '<S2>/TofReset' */

  /* Outputs for Atomic SubSystem: '<S2>/Filter' */
  /* RelationalOperator: '<S3>/Relational Operator' incorporates:
   *  Constant: '<S3>/Constant'
   */
  rtb_trigger_LVRT_l = (GridStat_B->BusInput.rTi_Filt_factorNoffsetCorr > 0.0F);

  /* Logic: '<S3>/Logical Operator' incorporates:
   *  Logic: '<S3>/Logical Operator1'
   */
  rtb_LogicalOperator_b = (GridStat_B->TofReset.LogicalOperator1 ||
    (!rtb_trigger_LVRT_l));

  /* DiscreteIntegrator: '<S3>/Discrete-Time Integrator' */
  if (rtb_LogicalOperator_b || (GridStat_DWork->DiscreteTimeIntegrator_PrevRe_g
       != 0)) {
    GridStat_DWork->DiscreteTimeIntegrator_DSTATE = 0.0;
  }

  /* Switch: '<S3>/Switch' incorporates:
   *  Constant: '<S2>/Constant12'
   *  DiscreteIntegrator: '<S3>/Discrete-Time Integrator'
   */
  if (rtb_trigger_LVRT_l) {
    rtb_Switch = GridStat_DWork->DiscreteTimeIntegrator_DSTATE;
  } else {
    rtb_Switch = 1.0;
  }

  /* End of Switch: '<S3>/Switch' */

  /* Switch: '<S9>/Switch' incorporates:
   *  Abs: '<S9>/Abs'
   *  RelationalOperator: '<S9>/Relational Operator'
   */
  if (2.22044605E-16F >= (real32_T)fabs
      (GridStat_B->BusInput.rTi_Filt_factorNoffsetCorr)) {
    rtb_Product5 = 2.22044605E-16F;
  } else {
    rtb_Product5 = GridStat_B->BusInput.rTi_Filt_factorNoffsetCorr;
  }

  /* End of Switch: '<S9>/Switch' */

  /* Update for DiscreteIntegrator: '<S3>/Discrete-Time Integrator' incorporates:
   *  Constant: '<S2>/Constant12'
   *  Product: '<S3>/Divide4'
   *  Sum: '<S3>/Sum4'
   */
  GridStat_DWork->DiscreteTimeIntegrator_DSTATE += (1.0 -
    GridStat_DWork->DiscreteTimeIntegrator_DSTATE) / rtb_Product5 * 0.01;
  GridStat_DWork->DiscreteTimeIntegrator_PrevRe_g = (int8_T)
    rtb_LogicalOperator_b;

  /* End of Outputs for SubSystem: '<S2>/Filter' */

  /* Logic: '<S2>/Logical Operator4' */
  rtb_trigger_LVRT_l = !rtb_AND;

  /* Delay: '<S2>/IslandDetected' */
  GridStat_DWork->icLoad = ((((GridStat_PrevZCSigState->IslandDetected_Reset_ZCE
    == 1) != (int32_T)GridStat_B->BusInput2.bReset) &&
    (GridStat_PrevZCSigState->IslandDetected_Reset_ZCE != 3)) ||
    GridStat_B->BusInput2.bReset || GridStat_DWork->icLoad);
  GridStat_PrevZCSigState->IslandDetected_Reset_ZCE =
    GridStat_B->BusInput2.bReset;
  GridStat_DWork->IslandDetected_DSTATE = ((!GridStat_DWork->icLoad) &&
    GridStat_DWork->IslandDetected_DSTATE);

  /* Switch: '<S2>/Switch1' incorporates:
   *  Delay: '<S2>/IslandDetected'
   *  Logic: '<S2>/Logical Operator6'
   */
  if (rtb_trigger_LVRT_l || rtb_LogicalOperator3) {
    rtb_AND = rtb_LogicalOperator3;
  } else {
    rtb_AND = GridStat_DWork->IslandDetected_DSTATE;
  }

  /* End of Switch: '<S2>/Switch1' */

  /* Logic: '<Root>/Logical Operator' incorporates:
   *  Logic: '<S2>/Logical Operator2'
   */
  GridStat_Y->Out.bGridStatus = ((!rtb_trigger_LVRT_l) && (!rtb_AND));

  /* Product: '<S2>/Product' */
  u0 = rtb_Switch * GridStat_B->BusInput2.rN_F_Offset_Norm;

  /* MinMax: '<S2>/MinMax1' */
  if (u0 <= GridStat_B->BusInput2.rN_F_Offset_Norm) {
    /* BusCreator: '<Root>/Bus Creator1' incorporates:
     *  DataTypeConversion: '<Root>/Data Type Conversion1'
     *  Outport: '<Root>/Out'
     */
    GridStat_Y->Out.rN_F_Offset_Norm_corr = (real32_T)u0;
  } else {
    /* BusCreator: '<Root>/Bus Creator1' incorporates:
     *  Outport: '<Root>/Out'
     */
    GridStat_Y->Out.rN_F_Offset_Norm_corr =
      GridStat_B->BusInput2.rN_F_Offset_Norm;
  }

  /* End of MinMax: '<S2>/MinMax1' */

  /* BusCreator generated from: '<Root>/dbg' incorporates:
   *  DataTypeConversion: '<S2>/Data Type Conversion1'
   *  MATLAB Function: '<S5>/Grid Observer'
   *  Outport: '<Root>/dbg'
   */
  GridStat_Y->dbg.rProt_norm = rtb_Saturation;
  GridStat_Y->dbg.bDetSpeedRise =
    GridStat_B->TpDetNabsProtTrigger.LogicalOperator1;
  GridStat_Y->dbg.bDetIslandVPN = GridStat_B->TpDetVPNTrigger.LogicalOperator1;
  GridStat_Y->dbg.trigger_Nabs = rtb_RelationalOperator;
  GridStat_Y->dbg.trigger_Prot = rtb_LogicalOperator_i;
  GridStat_Y->dbg.trigger_PU = rtb_trigger_PU;
  GridStat_Y->dbg.trigger_N = rtb_trigger_N;
  GridStat_Y->dbg.trigger_U = rtb_trigger_U;
  GridStat_Y->dbg.trigger_P = rtb_trigger_P;
  GridStat_Y->dbg.trigger_VS = GridStat_B->BusInput2.bVectorShift;
  GridStat_Y->dbg.block_LVRT_VPN = rtb_Switch6;
  GridStat_Y->dbg.trigger_LVRT_NoDelay = rtb_RelationalOperator3_dy;
  GridStat_Y->dbg.rCorrFac_rN_set_Norm = (real32_T)rtb_Switch;
  GridStat_Y->dbg.block_LVRT_speedAbs = rtb_RelationalOperator3;
  GridStat_Y->dbg.bDetGridObserver = rtb_RelationalOperator_b;
  for (i = 0; i < 9; i++) {
    GridStat_Y->dbg.ru_obs[i] = 0.0F;
    GridStat_Y->dbg.ru_obs_strong[i] = 0.0F;
    GridStat_Y->dbg.ru_obs3[i] = 0.0F;
  }

  GridStat_Y->dbg.ry_obs[0] = 0.0F;
  GridStat_Y->dbg.ry_obs[1] = 0.0F;
  for (i = 0; i < 5; i++) {
    GridStat_Y->dbg.rx_obs[i] = 0.0F;
    GridStat_Y->dbg.rx_obs_strong[i] = 0.0F;
    GridStat_Y->dbg.rx_obs3[i] = 0.0F;
    GridStat_Y->dbg.rcorr[i] = 0.0F;
    GridStat_Y->dbg.rcorr_strong[i] = 0.0F;
    GridStat_Y->dbg.rcorr3[i] = 0.0F;
  }

  /* End of BusCreator generated from: '<Root>/dbg' */

  /* S-Function (bur_bus_out): '<Root>/Bus Output' incorporates:
   *  Outport: '<Root>/Out'
   */
  inst->Out = GridStat_Y->Out;

  /* BusCreator generated from: '<Root>/Bus Output1' incorporates:
   *  DataTypeConversion: '<S2>/Data Type Conversion1'
   *  MATLAB Function: '<S5>/Grid Observer'
   */
  GridStat_B->BusConversion_InsertedFor_BusOu.rProt_norm = rtb_Saturation;
  GridStat_B->BusConversion_InsertedFor_BusOu.bDetSpeedRise =
    GridStat_B->TpDetNabsProtTrigger.LogicalOperator1;
  GridStat_B->BusConversion_InsertedFor_BusOu.bDetIslandVPN =
    GridStat_B->TpDetVPNTrigger.LogicalOperator1;
  GridStat_B->BusConversion_InsertedFor_BusOu.trigger_Nabs =
    rtb_RelationalOperator;
  GridStat_B->BusConversion_InsertedFor_BusOu.trigger_Prot =
    rtb_LogicalOperator_i;
  GridStat_B->BusConversion_InsertedFor_BusOu.trigger_PU = rtb_trigger_PU;
  GridStat_B->BusConversion_InsertedFor_BusOu.trigger_N = rtb_trigger_N;
  GridStat_B->BusConversion_InsertedFor_BusOu.trigger_U = rtb_trigger_U;
  GridStat_B->BusConversion_InsertedFor_BusOu.trigger_P = rtb_trigger_P;
  GridStat_B->BusConversion_InsertedFor_BusOu.trigger_VS =
    GridStat_B->BusInput2.bVectorShift;
  GridStat_B->BusConversion_InsertedFor_BusOu.block_LVRT_VPN = rtb_Switch6;
  GridStat_B->BusConversion_InsertedFor_BusOu.trigger_LVRT_NoDelay =
    rtb_RelationalOperator3_dy;
  GridStat_B->BusConversion_InsertedFor_BusOu.rCorrFac_rN_set_Norm = (real32_T)
    rtb_Switch;
  GridStat_B->BusConversion_InsertedFor_BusOu.block_LVRT_speedAbs =
    rtb_RelationalOperator3;
  GridStat_B->BusConversion_InsertedFor_BusOu.bDetGridObserver =
    rtb_RelationalOperator_b;
  for (i = 0; i < 9; i++) {
    GridStat_B->BusConversion_InsertedFor_BusOu.ru_obs[i] = 0.0F;
    GridStat_B->BusConversion_InsertedFor_BusOu.ru_obs_strong[i] = 0.0F;
    GridStat_B->BusConversion_InsertedFor_BusOu.ru_obs3[i] = 0.0F;
  }

  GridStat_B->BusConversion_InsertedFor_BusOu.ry_obs[0] = 0.0F;
  GridStat_B->BusConversion_InsertedFor_BusOu.ry_obs[1] = 0.0F;
  for (i = 0; i < 5; i++) {
    GridStat_B->BusConversion_InsertedFor_BusOu.rx_obs[i] = 0.0F;
    GridStat_B->BusConversion_InsertedFor_BusOu.rx_obs_strong[i] = 0.0F;
    GridStat_B->BusConversion_InsertedFor_BusOu.rx_obs3[i] = 0.0F;
    GridStat_B->BusConversion_InsertedFor_BusOu.rcorr[i] = 0.0F;
    GridStat_B->BusConversion_InsertedFor_BusOu.rcorr_strong[i] = 0.0F;
    GridStat_B->BusConversion_InsertedFor_BusOu.rcorr3[i] = 0.0F;
  }

  /* End of BusCreator generated from: '<Root>/Bus Output1' */

  /* S-Function (bur_bus_out): '<Root>/Bus Output1' */
  inst->Dbg = GridStat_B->BusConversion_InsertedFor_BusOu;

  /* S-Function (bur_bus_in): '<Root>/Bus Input1' */
  GridStat_B->BusInput1 = inst->Perm;

  /* UnitDelay: '<S1>/Unit Delay' */
  GridStat_B->UnitDelay = GridStat_DWork->UnitDelay_DSTATE;

  /* S-Function (bur_out): '<Root>/Bus Output2' */
  inst->Version = GridStat_B->UnitDelay;
  for (i = 0; i < 9; i++) {
    /* Update for S-Function (sfix_udelay): '<S8>/Tapped Delay' */
    GridStat_DWork->TappedDelay_X[9 - i] = GridStat_DWork->TappedDelay_X[8 - i];

    /* Update for S-Function (sfix_udelay): '<S8>/Tapped Delay1' */
    GridStat_DWork->TappedDelay1_X[9 - i] = GridStat_DWork->TappedDelay1_X[8 - i];

    /* Update for S-Function (sfix_udelay): '<S8>/Tapped Delay2' */
    GridStat_DWork->TappedDelay2_X[9 - i] = GridStat_DWork->TappedDelay2_X[8 - i];

    /* Update for S-Function (sfix_udelay): '<S5>/Tapped Delay' */
    GridStat_DWork->TappedDelay_X_l[9 - i] = GridStat_DWork->TappedDelay_X_l[8 -
      i];

    /* Update for S-Function (sfix_udelay): '<S5>/Tapped Delay2' */
    GridStat_DWork->TappedDelay2_X_b[9 - i] = GridStat_DWork->TappedDelay2_X_b[8
      - i];

    /* Update for S-Function (sfix_udelay): '<S5>/Tapped Delay3' */
    GridStat_DWork->TappedDelay3_X[9 - i] = GridStat_DWork->TappedDelay3_X[8 - i];

    /* Update for S-Function (sfix_udelay): '<S5>/Tapped Delay5' */
    GridStat_DWork->TappedDelay5_X[9 - i] = GridStat_DWork->TappedDelay5_X[8 - i];

    /* Update for S-Function (sfix_udelay): '<S5>/Tapped Delay4' */
    GridStat_DWork->TappedDelay4_X[9 - i] = GridStat_DWork->TappedDelay4_X[8 - i];

    /* Update for S-Function (sfix_udelay): '<S5>/Tapped Delay1' */
    GridStat_DWork->TappedDelay1_X_m[9 - i] = GridStat_DWork->TappedDelay1_X_m[8
      - i];
  }

  /* Update for S-Function (sfix_udelay): '<S8>/Tapped Delay' */
  GridStat_DWork->TappedDelay_X[0] = GridStat_B->BusInput2.rU_norm;

  /* Update for S-Function (sfix_udelay): '<S8>/Tapped Delay1' */
  GridStat_DWork->TappedDelay1_X[0] = GridStat_B->BusInput2.rP_norm;

  /* Update for S-Function (sfix_udelay): '<S8>/Tapped Delay2' */
  GridStat_DWork->TappedDelay2_X[0] = GridStat_B->BusInput2.rN_engAct;

  /* Update for S-Function (sfix_udelay): '<S5>/Tapped Delay' */
  GridStat_DWork->TappedDelay_X_l[0] = GridStat_B->BusInput2.rp2s_norm;

  /* Update for S-Function (sfix_udelay): '<S5>/Tapped Delay2' */
  GridStat_DWork->TappedDelay2_X_b[0] = GridStat_B->BusInput2.rP_norm;

  /* Update for S-Function (sfix_udelay): '<S5>/Tapped Delay3' */
  GridStat_DWork->TappedDelay3_X[0] = GridStat_B->BusInput2.rN_engAct;

  /* Update for S-Function (sfix_udelay): '<S5>/Tapped Delay5' */
  GridStat_DWork->TappedDelay5_X[0] = GridStat_B->BusInput2.rQ_norm;

  /* Update for S-Function (sfix_udelay): '<S5>/Tapped Delay4' */
  GridStat_DWork->TappedDelay4_X[0] = GridStat_B->BusInput2.rU_norm;

  /* Update for S-Function (sfix_udelay): '<S5>/Tapped Delay1' */
  GridStat_DWork->TappedDelay1_X_m[0] = GridStat_B->BusInput2.rUexc_norm;

  /* Update for Delay: '<S2>/IslandDetected' */
  GridStat_DWork->icLoad = false;
  GridStat_DWork->IslandDetected_DSTATE = rtb_AND;

  /* Update for UnitDelay: '<S1>/Unit Delay' */
  GridStat_DWork->UnitDelay_DSTATE = 202U;
}

/* Model initialize function */
void GridStat_initialize(RT_MODEL_GridStat *const GridStat_M, struct fGridStat* inst)
{
  struct D_Work_GridStat *GridStat_DWork = GridStat_M->dwork;
  struct PrevZCSigStates_GridStat *GridStat_PrevZCSigState = GridStat_M->prevZCSigState;
  GridStat_PrevZCSigState->IslandDetected_Reset_ZCE = UNINITIALIZED_ZCSIG;

  /* InitializeConditions for Delay: '<S2>/IslandDetected' */
  GridStat_DWork->icLoad = true;

  /* SystemInitialize for Atomic SubSystem: '<S2>/TofMcbFb' */
  GridStat_TofLvrtWeakBlk1_Init(&GridStat_DWork->TofMcbFb, inst);

  /* End of SystemInitialize for SubSystem: '<S2>/TofMcbFb' */

  /* SystemInitialize for Atomic SubSystem: '<S4>/TpNabsTrigger' */
  GridS_TpDetNabsProtTrigger_Init(&GridStat_DWork->TpNabsTrigger, inst);

  /* End of SystemInitialize for SubSystem: '<S4>/TpNabsTrigger' */

  /* SystemInitialize for Atomic SubSystem: '<S4>/Speed_filter' */
  /* InitializeConditions for DiscreteIntegrator: '<S11>/Discrete-Time Integrator' */
  GridStat_DWork->DiscreteTimeIntegrator_IC_LOADI = 1U;

  /* End of SystemInitialize for SubSystem: '<S4>/Speed_filter' */

  /* SystemInitialize for Atomic SubSystem: '<S4>/TpProtTrigger' */
  GridS_TpDetNabsProtTrigger_Init(&GridStat_DWork->TpProtTrigger, inst);

  /* End of SystemInitialize for SubSystem: '<S4>/TpProtTrigger' */

  /* SystemInitialize for Atomic SubSystem: '<S4>/TpLvrtBlockHold1' */
  GridS_TpDetNabsProtTrigger_Init(&GridStat_DWork->TpLvrtBlockHold1, inst);

  /* End of SystemInitialize for SubSystem: '<S4>/TpLvrtBlockHold1' */

  /* SystemInitialize for Atomic SubSystem: '<S4>/TofLvrtWeakBlk1' */
  GridStat_TofLvrtWeakBlk1_Init(&GridStat_DWork->TofLvrtWeakBlk1, inst);

  /* End of SystemInitialize for SubSystem: '<S4>/TofLvrtWeakBlk1' */

  /* SystemInitialize for Atomic SubSystem: '<S4>/TpLvrtTrigHold1' */
  GridS_TpDetNabsProtTrigger_Init(&GridStat_DWork->TpLvrtTrigHold1, inst);

  /* End of SystemInitialize for SubSystem: '<S4>/TpLvrtTrigHold1' */

  /* SystemInitialize for Atomic SubSystem: '<S4>/TpDetNabsProtTrigger' */
  GridS_TpDetNabsProtTrigger_Init(&GridStat_DWork->TpDetNabsProtTrigger, inst);

  /* End of SystemInitialize for SubSystem: '<S4>/TpDetNabsProtTrigger' */

  /* SystemInitialize for Atomic SubSystem: '<S8>/TofLvrtWeakBlk2' */
  GridStat_TofLvrtWeakBlk1_Init(&GridStat_DWork->TofLvrtWeakBlk2, inst);

  /* End of SystemInitialize for SubSystem: '<S8>/TofLvrtWeakBlk2' */

  /* SystemInitialize for Atomic SubSystem: '<S8>/TpLvrtTrigHold2' */
  GridS_TpDetNabsProtTrigger_Init(&GridStat_DWork->TpLvrtTrigHold2, inst);

  /* End of SystemInitialize for SubSystem: '<S8>/TpLvrtTrigHold2' */

  /* SystemInitialize for Atomic SubSystem: '<S8>/TofAfterFRT' */
  GridStat_TofLvrtWeakBlk1_Init(&GridStat_DWork->TofAfterFRT, inst);

  /* End of SystemInitialize for SubSystem: '<S8>/TofAfterFRT' */

  /* SystemInitialize for Atomic SubSystem: '<S8>/TpUTrigger' */
  GridS_TpDetNabsProtTrigger_Init(&GridStat_DWork->TpUTrigger, inst);

  /* End of SystemInitialize for SubSystem: '<S8>/TpUTrigger' */

  /* SystemInitialize for Atomic SubSystem: '<S8>/TpPTrigger' */
  GridS_TpDetNabsProtTrigger_Init(&GridStat_DWork->TpPTrigger, inst);

  /* End of SystemInitialize for SubSystem: '<S8>/TpPTrigger' */

  /* SystemInitialize for Atomic SubSystem: '<S8>/TP_PU_trigger' */
  GridS_TpDetNabsProtTrigger_Init(&GridStat_DWork->TP_PU_trigger, inst);

  /* End of SystemInitialize for SubSystem: '<S8>/TP_PU_trigger' */

  /* SystemInitialize for Atomic SubSystem: '<S8>/TpNTrigger' */
  GridS_TpDetNabsProtTrigger_Init(&GridStat_DWork->TpNTrigger, inst);

  /* End of SystemInitialize for SubSystem: '<S8>/TpNTrigger' */

  /* SystemInitialize for Atomic SubSystem: '<S8>/TpLvrtBlockHold2' */
  GridS_TpDetNabsProtTrigger_Init(&GridStat_DWork->TpLvrtBlockHold2, inst);

  /* End of SystemInitialize for SubSystem: '<S8>/TpLvrtBlockHold2' */

  /* SystemInitialize for Atomic SubSystem: '<S8>/TpDetVPNTrigger' */
  GridS_TpDetNabsProtTrigger_Init(&GridStat_DWork->TpDetVPNTrigger, inst);

  /* End of SystemInitialize for SubSystem: '<S8>/TpDetVPNTrigger' */

  /* SystemInitialize for Atomic SubSystem: '<S2>/TofReset' */
  GridStat_TofLvrtWeakBlk1_Init(&GridStat_DWork->TofReset, inst);

  /* End of SystemInitialize for SubSystem: '<S2>/TofReset' */
}

/* Model terminate function */
void GridStat_terminate(RT_MODEL_GridStat *const GridStat_M, struct fGridStat* inst)
{
  /* (no terminate code required) */
  UNUSED_PARAMETER(GridStat_M);
}

/*======================== TOOL VERSION INFORMATION ==========================*
 * MATLAB 9.11 (R2021b)14-May-2021                                            *
 * Simulink 10.4 (R2021b)14-May-2021                                          *
 * Simulink Coder 9.6 (R2021b)14-May-2021                                     *
 * Embedded Coder 7.7 (R2021b)14-May-2021                                     *
 * Stateflow 10.5 (R2021b)14-May-2021                                         *
 *============================================================================*/

/*======================= LICENSE IN USE INFORMATION =========================*
 * matlab                                                                     *
 * matlab_coder                                                               *
 * real-time_workshop                                                         *
 * rtw_embedded_coder                                                         *
 * simulink                                                                   *
 *============================================================================*/
```

#### GridStat.h
```c
/********************************************************************
 * COPYRIGHT -- B&R Industrial Automation GmbH
 ********************************************************************
 * Program: GridStat
 * File: GridStat.h
 * Author: 105055527
 * Last modified by: cadm_kafkama00
 * Created: Mon Sep 05 18:14:57 2016
 * Last modified: Tue Nov 26 15:54:38 2024
 * Model Version: 2.02
 * Description: Detection Algorithm for grid connection.

   HISTORY:
   V1.00  24.07.2020 Keller   created
   V1.01  07.08.2020 Huber  included function block from simulation
   V1.02  29.04.2021 Denk   VectorShift and LVRT function added
   V1.03  31.01.2022 Keller  add input for GCB_On

   V2.00  10.08.2023 Walch  Revision of parametrization, sensitivity and FRT selectivity
   V2.01  22.11.2023 Walch  Include grid observer
   10.01.2024 Walch  Include TP LVRT hold time for weak LVRT blocking
   V2.02  25.11.2024 Walch  Update grid observer for SS mains parallel vs. island plausibility check
 * modified Comment:
 ********************************************************************
 * Header for program GridStat
 ********************************************************************
 * Generated with B&R Automation Studio Target for Simulink V6.7.1
 * (ERT based)
 ********************************************************************/

#ifndef RTW_HEADER_GridStat_h_
#define RTW_HEADER_GridStat_h_
#include <math.h>
#ifndef GridStat_COMMON_INCLUDES_
#define GridStat_COMMON_INCLUDES_
#include "rtwtypes.h"
#include "zero_crossing_types.h"
#endif                                 /* GridStat_COMMON_INCLUDES_ */

#include "GridStat_types.h"
#include "lGridStat.h"
/* Beginning of Dynamic TypeDefs: */
/* End of Dynamic TypeDefs: */
#ifndef MIN
#define MIN(a,b)	((a) < (b) ? (a) : (b))
#endif

#ifndef MAX
#define MAX(a,b)	((a) > (b) ? (a) : (b))
#endif

#ifndef AST_ROUND
#define AST_ROUND(x) ((x)>=0?(long long)((x)+0.5):(long long)((x)-0.5))
#endif

#include "rt_defines.h"

/* Macros for accessing real-time model data structure */
#ifndef rtmGetBlockIO
#define rtmGetBlockIO(rtm)             ((rtm)->blockIO)
#endif

#ifndef rtmSetBlockIO
#define rtmSetBlockIO(rtm, val)        ((rtm)->blockIO = (val))
#endif

#ifndef rtmGetPrevZCSigState
#define rtmGetPrevZCSigState(rtm)      ((rtm)->prevZCSigState)
#endif

#ifndef rtmSetPrevZCSigState
#define rtmSetPrevZCSigState(rtm, val) ((rtm)->prevZCSigState = (val))
#endif

#ifndef rtmGetRootDWork
#define rtmGetRootDWork(rtm)           ((rtm)->dwork)
#endif

#ifndef rtmSetRootDWork
#define rtmSetRootDWork(rtm, val)      ((rtm)->dwork = (val))
#endif

#ifndef rtmGetY
#define rtmGetY(rtm)                   ((rtm)->outputs)
#endif

#ifndef rtmSetY
#define rtmSetY(rtm, val)              ((rtm)->outputs = (val))
#endif

#ifndef rtmGetErrorStatus
#define rtmGetErrorStatus(rtm)         ((rtm)->errorStatus)
#endif

#ifndef rtmSetErrorStatus
#define rtmSetErrorStatus(rtm, val)    ((rtm)->errorStatus = (val))
#endif

#ifndef MIN
#define MIN(a,b)                       ((a) < (b) ? (a) : (b))
#endif

#ifndef MAX
#define MAX(a,b)                       ((a) > (b) ? (a) : (b))
#endif

#ifndef AST_ROUND
#define AST_ROUND(x)                   ((x)>=0?(long long)((x)+0.5):(long long)((x)-0.5))
#endif

/* user code (top of header file) */
/***************************************************************************************************
 * COPYRIGHT -- INNIO Jenbacher GmbH & CO OG
 ****************************************************************************************************
 * Program:            GridStat
 * Author:             cadm_kafkama00
 * Created:            26.11.2024 15:54
 ****************************************************************************************************
 * MODEL INFORMATION
 ****************************************************************************************************
 * Model Name:         C:\Users\kafkama00\Documents\Git\JenCtrLib\Controllers\GridStatusDetection\GridStat.slx
 * Model Version:      2.02
 * Simulink Version:   R2021b
 * B&R Target:         V6.7.1
 * Description:        Detection Algorithm for grid connection.
 *
 *                     HISTORY:
 *                     V1.00  24.07.2020 Keller   created
 *                     V1.01  07.08.2020 Huber  included function block from simulation
 *                     V1.02  29.04.2021 Denk   VectorShift and LVRT function added
 *                     V1.03  31.01.2022 Keller  add input for GCB_On
 *
 *                     V2.00  10.08.2023 Walch  Revision of parametrization, sensitivity and FRT selectivity
 *                     V2.01  22.11.2023 Walch  Include grid observer
 *                                10.01.2024 Walch  Include TP LVRT hold time for weak LVRT blocking
 *                     V2.02  25.11.2024 Walch  Update grid observer for SS mains parallel vs. island plausibility check
 ****************************************************************************************************
 * Last Modified By:   walchin00
 * Last Modified Date: Mon Nov 25 17:05:58 2024
 ****************************************************************************************************/

/* Block signals for system '<S4>/TofLvrtWeakBlk1' */

/* Block states (default storage) for system '<S4>/TofLvrtWeakBlk1' */

/* Block signals for system '<S4>/TpDetNabsProtTrigger' */

/* Block states (default storage) for system '<S4>/TpDetNabsProtTrigger' */

/* Block signals (default storage) */

/* Block states (default storage) for system '<Root>' */

/* Zero-crossing (trigger) state */

/* External outputs (root outports fed by signals with default storage) */

/* Real-time Model Data Structure */

/* Model entry point functions */
extern void GridStat_initialize(RT_MODEL_GridStat *const GridStat_M, struct fGridStat* inst);
extern void GridStat_step(RT_MODEL_GridStat *const GridStat_M, struct fGridStat* inst);
extern void GridStat_terminate(RT_MODEL_GridStat *const GridStat_M, struct fGridStat* inst);

/*-
 * The generated code includes comments that allow you to trace directly
 * back to the appropriate location in the model.  The basic format
 * is <system>/block_name, where system is the system number (uniquely
 * assigned by Simulink) and block_name is the name of the block.
 *
 * Use the MATLAB hilite_system command to trace the generated code back
 * to the model.  For example,
 *
 * hilite_system('<S3>')    - opens system 3
 * hilite_system('<S3>/Kp') - opens and selects block Kp which resides in S3
 *
 * Here is the system hierarchy for this model
 *
 * '<Root>' : 'GridStat'
 * '<S1>'   : 'GridStat/Info1'
 * '<S2>'   : 'GridStat/detection + correction: transition to Island'
 * '<S3>'   : 'GridStat/detection + correction: transition to Island/Filter'
 * '<S4>'   : 'GridStat/detection + correction: transition to Island/N//Prot Detection'
 * '<S5>'   : 'GridStat/detection + correction: transition to Island/Smooth Detection'
 * '<S6>'   : 'GridStat/detection + correction: transition to Island/TofMcbFb'
 * '<S7>'   : 'GridStat/detection + correction: transition to Island/TofReset'
 * '<S8>'   : 'GridStat/detection + correction: transition to Island/VPN Detection'
 * '<S9>'   : 'GridStat/detection + correction: transition to Island/Filter/Divisor'
 * '<S10>'  : 'GridStat/detection + correction: transition to Island/Filter/Divisor/Data Type Conversion Inherited'
 * '<S11>'  : 'GridStat/detection + correction: transition to Island/N//Prot Detection/Speed_filter'
 * '<S12>'  : 'GridStat/detection + correction: transition to Island/N//Prot Detection/TofLvrtWeakBlk1'
 * '<S13>'  : 'GridStat/detection + correction: transition to Island/N//Prot Detection/TpDetNabsProtTrigger'
 * '<S14>'  : 'GridStat/detection + correction: transition to Island/N//Prot Detection/TpLvrtBlockHold1'
 * '<S15>'  : 'GridStat/detection + correction: transition to Island/N//Prot Detection/TpLvrtTrigHold1'
 * '<S16>'  : 'GridStat/detection + correction: transition to Island/N//Prot Detection/TpNabsTrigger'
 * '<S17>'  : 'GridStat/detection + correction: transition to Island/N//Prot Detection/TpProtTrigger'
 * '<S18>'  : 'GridStat/detection + correction: transition to Island/N//Prot Detection/Speed_filter/Divisor'
 * '<S19>'  : 'GridStat/detection + correction: transition to Island/N//Prot Detection/Speed_filter/Divisor/Data Type Conversion Inherited'
 * '<S20>'  : 'GridStat/detection + correction: transition to Island/N//Prot Detection/TofLvrtWeakBlk1/Data Type Conversion Inherited'
 * '<S21>'  : 'GridStat/detection + correction: transition to Island/N//Prot Detection/TpDetNabsProtTrigger/Compare To Zero'
 * '<S22>'  : 'GridStat/detection + correction: transition to Island/N//Prot Detection/TpDetNabsProtTrigger/Enabled Subsystem'
 * '<S23>'  : 'GridStat/detection + correction: transition to Island/N//Prot Detection/TpDetNabsProtTrigger/Enabled Subsystem1'
 * '<S24>'  : 'GridStat/detection + correction: transition to Island/N//Prot Detection/TpDetNabsProtTrigger/Rate Limiter'
 * '<S25>'  : 'GridStat/detection + correction: transition to Island/N//Prot Detection/TpDetNabsProtTrigger/Rate Limiter/Saturation Dynamic'
 * '<S26>'  : 'GridStat/detection + correction: transition to Island/N//Prot Detection/TpLvrtBlockHold1/Compare To Zero'
 * '<S27>'  : 'GridStat/detection + correction: transition to Island/N//Prot Detection/TpLvrtBlockHold1/Enabled Subsystem'
 * '<S28>'  : 'GridStat/detection + correction: transition to Island/N//Prot Detection/TpLvrtBlockHold1/Enabled Subsystem1'
 * '<S29>'  : 'GridStat/detection + correction: transition to Island/N//Prot Detection/TpLvrtBlockHold1/Rate Limiter'
 * '<S30>'  : 'GridStat/detection + correction: transition to Island/N//Prot Detection/TpLvrtBlockHold1/Rate Limiter/Saturation Dynamic'
 * '<S31>'  : 'GridStat/detection + correction: transition to Island/N//Prot Detection/TpLvrtTrigHold1/Compare To Zero'
 * '<S32>'  : 'GridStat/detection + correction: transition to Island/N//Prot Detection/TpLvrtTrigHold1/Enabled Subsystem'
 * '<S33>'  : 'GridStat/detection + correction: transition to Island/N//Prot Detection/TpLvrtTrigHold1/Enabled Subsystem1'
 * '<S34>'  : 'GridStat/detection + correction: transition to Island/N//Prot Detection/TpLvrtTrigHold1/Rate Limiter'
 * '<S35>'  : 'GridStat/detection + correction: transition to Island/N//Prot Detection/TpLvrtTrigHold1/Rate Limiter/Saturation Dynamic'
 * '<S36>'  : 'GridStat/detection + correction: transition to Island/N//Prot Detection/TpNabsTrigger/Compare To Zero'
 * '<S37>'  : 'GridStat/detection + correction: transition to Island/N//Prot Detection/TpNabsTrigger/Enabled Subsystem'
 * '<S38>'  : 'GridStat/detection + correction: transition to Island/N//Prot Detection/TpNabsTrigger/Enabled Subsystem1'
 * '<S39>'  : 'GridStat/detection + correction: transition to Island/N//Prot Detection/TpNabsTrigger/Rate Limiter'
 * '<S40>'  : 'GridStat/detection + correction: transition to Island/N//Prot Detection/TpNabsTrigger/Rate Limiter/Saturation Dynamic'
 * '<S41>'  : 'GridStat/detection + correction: transition to Island/N//Prot Detection/TpProtTrigger/Compare To Zero'
 * '<S42>'  : 'GridStat/detection + correction: transition to Island/N//Prot Detection/TpProtTrigger/Enabled Subsystem'
 * '<S43>'  : 'GridStat/detection + correction: transition to Island/N//Prot Detection/TpProtTrigger/Enabled Subsystem1'
 * '<S44>'  : 'GridStat/detection + correction: transition to Island/N//Prot Detection/TpProtTrigger/Rate Limiter'
 * '<S45>'  : 'GridStat/detection + correction: transition to Island/N//Prot Detection/TpProtTrigger/Rate Limiter/Saturation Dynamic'
 * '<S46>'  : 'GridStat/detection + correction: transition to Island/Smooth Detection/Divisor'
 * '<S47>'  : 'GridStat/detection + correction: transition to Island/Smooth Detection/Divisor1'
 * '<S48>'  : 'GridStat/detection + correction: transition to Island/Smooth Detection/Divisor2'
 * '<S49>'  : 'GridStat/detection + correction: transition to Island/Smooth Detection/Divisor3'
 * '<S50>'  : 'GridStat/detection + correction: transition to Island/Smooth Detection/Divisor4'
 * '<S51>'  : 'GridStat/detection + correction: transition to Island/Smooth Detection/Divisor5'
 * '<S52>'  : 'GridStat/detection + correction: transition to Island/Smooth Detection/Grid Observer'
 * '<S53>'  : 'GridStat/detection + correction: transition to Island/Smooth Detection/Divisor/Data Type Conversion Inherited'
 * '<S54>'  : 'GridStat/detection + correction: transition to Island/Smooth Detection/Divisor1/Data Type Conversion Inherited'
 * '<S55>'  : 'GridStat/detection + correction: transition to Island/Smooth Detection/Divisor2/Data Type Conversion Inherited'
 * '<S56>'  : 'GridStat/detection + correction: transition to Island/Smooth Detection/Divisor3/Data Type Conversion Inherited'
 * '<S57>'  : 'GridStat/detection + correction: transition to Island/Smooth Detection/Divisor4/Data Type Conversion Inherited'
 * '<S58>'  : 'GridStat/detection + correction: transition to Island/Smooth Detection/Divisor5/Data Type Conversion Inherited'
 * '<S59>'  : 'GridStat/detection + correction: transition to Island/TofMcbFb/Data Type Conversion Inherited'
 * '<S60>'  : 'GridStat/detection + correction: transition to Island/TofReset/Data Type Conversion Inherited'
 * '<S61>'  : 'GridStat/detection + correction: transition to Island/VPN Detection/TP_PU_trigger'
 * '<S62>'  : 'GridStat/detection + correction: transition to Island/VPN Detection/TofAfterFRT'
 * '<S63>'  : 'GridStat/detection + correction: transition to Island/VPN Detection/TofLvrtWeakBlk2'
 * '<S64>'  : 'GridStat/detection + correction: transition to Island/VPN Detection/TpDetVPNTrigger'
 * '<S65>'  : 'GridStat/detection + correction: transition to Island/VPN Detection/TpLvrtBlockHold2'
 * '<S66>'  : 'GridStat/detection + correction: transition to Island/VPN Detection/TpLvrtTrigHold2'
 * '<S67>'  : 'GridStat/detection + correction: transition to Island/VPN Detection/TpNTrigger'
 * '<S68>'  : 'GridStat/detection + correction: transition to Island/VPN Detection/TpPTrigger'
 * '<S69>'  : 'GridStat/detection + correction: transition to Island/VPN Detection/TpUTrigger'
 * '<S70>'  : 'GridStat/detection + correction: transition to Island/VPN Detection/TP_PU_trigger/Compare To Zero'
 * '<S71>'  : 'GridStat/detection + correction: transition to Island/VPN Detection/TP_PU_trigger/Enabled Subsystem'
 * '<S72>'  : 'GridStat/detection + correction: transition to Island/VPN Detection/TP_PU_trigger/Enabled Subsystem1'
 * '<S73>'  : 'GridStat/detection + correction: transition to Island/VPN Detection/TP_PU_trigger/Rate Limiter'
 * '<S74>'  : 'GridStat/detection + correction: transition to Island/VPN Detection/TP_PU_trigger/Rate Limiter/Saturation Dynamic'
 * '<S75>'  : 'GridStat/detection + correction: transition to Island/VPN Detection/TofAfterFRT/Data Type Conversion Inherited'
 * '<S76>'  : 'GridStat/detection + correction: transition to Island/VPN Detection/TofLvrtWeakBlk2/Data Type Conversion Inherited'
 * '<S77>'  : 'GridStat/detection + correction: transition to Island/VPN Detection/TpDetVPNTrigger/Compare To Zero'
 * '<S78>'  : 'GridStat/detection + correction: transition to Island/VPN Detection/TpDetVPNTrigger/Enabled Subsystem'
 * '<S79>'  : 'GridStat/detection + correction: transition to Island/VPN Detection/TpDetVPNTrigger/Enabled Subsystem1'
 * '<S80>'  : 'GridStat/detection + correction: transition to Island/VPN Detection/TpDetVPNTrigger/Rate Limiter'
 * '<S81>'  : 'GridStat/detection + correction: transition to Island/VPN Detection/TpDetVPNTrigger/Rate Limiter/Saturation Dynamic'
 * '<S82>'  : 'GridStat/detection + correction: transition to Island/VPN Detection/TpLvrtBlockHold2/Compare To Zero'
 * '<S83>'  : 'GridStat/detection + correction: transition to Island/VPN Detection/TpLvrtBlockHold2/Enabled Subsystem'
 * '<S84>'  : 'GridStat/detection + correction: transition to Island/VPN Detection/TpLvrtBlockHold2/Enabled Subsystem1'
 * '<S85>'  : 'GridStat/detection + correction: transition to Island/VPN Detection/TpLvrtBlockHold2/Rate Limiter'
 * '<S86>'  : 'GridStat/detection + correction: transition to Island/VPN Detection/TpLvrtBlockHold2/Rate Limiter/Saturation Dynamic'
 * '<S87>'  : 'GridStat/detection + correction: transition to Island/VPN Detection/TpLvrtTrigHold2/Compare To Zero'
 * '<S88>'  : 'GridStat/detection + correction: transition to Island/VPN Detection/TpLvrtTrigHold2/Enabled Subsystem'
 * '<S89>'  : 'GridStat/detection + correction: transition to Island/VPN Detection/TpLvrtTrigHold2/Enabled Subsystem1'
 * '<S90>'  : 'GridStat/detection + correction: transition to Island/VPN Detection/TpLvrtTrigHold2/Rate Limiter'
 * '<S91>'  : 'GridStat/detection + correction: transition to Island/VPN Detection/TpLvrtTrigHold2/Rate Limiter/Saturation Dynamic'
 * '<S92>'  : 'GridStat/detection + correction: transition to Island/VPN Detection/TpNTrigger/Compare To Zero'
 * '<S93>'  : 'GridStat/detection + correction: transition to Island/VPN Detection/TpNTrigger/Enabled Subsystem'
 * '<S94>'  : 'GridStat/detection + correction: transition to Island/VPN Detection/TpNTrigger/Enabled Subsystem1'
 * '<S95>'  : 'GridStat/detection + correction: transition to Island/VPN Detection/TpNTrigger/Rate Limiter'
 * '<S96>'  : 'GridStat/detection + correction: transition to Island/VPN Detection/TpNTrigger/Rate Limiter/Saturation Dynamic'
 * '<S97>'  : 'GridStat/detection + correction: transition to Island/VPN Detection/TpPTrigger/Compare To Zero'
 * '<S98>'  : 'GridStat/detection + correction: transition to Island/VPN Detection/TpPTrigger/Enabled Subsystem'
 * '<S99>'  : 'GridStat/detection + correction: transition to Island/VPN Detection/TpPTrigger/Enabled Subsystem1'
 * '<S100>' : 'GridStat/detection + correction: transition to Island/VPN Detection/TpPTrigger/Rate Limiter'
 * '<S101>' : 'GridStat/detection + correction: transition to Island/VPN Detection/TpPTrigger/Rate Limiter/Saturation Dynamic'
 * '<S102>' : 'GridStat/detection + correction: transition to Island/VPN Detection/TpUTrigger/Compare To Zero'
 * '<S103>' : 'GridStat/detection + correction: transition to Island/VPN Detection/TpUTrigger/Enabled Subsystem'
 * '<S104>' : 'GridStat/detection + correction: transition to Island/VPN Detection/TpUTrigger/Enabled Subsystem1'
 * '<S105>' : 'GridStat/detection + correction: transition to Island/VPN Detection/TpUTrigger/Rate Limiter'
 * '<S106>' : 'GridStat/detection + correction: transition to Island/VPN Detection/TpUTrigger/Rate Limiter/Saturation Dynamic'
 */
#endif                                 /* RTW_HEADER_GridStat_h_ */
```

#### GridStat_private.h
```c
/********************************************************************
 * COPYRIGHT -- B&R Industrial Automation GmbH
 ********************************************************************
 * Program: GridStat
 * File: GridStat_private.h
 * Author: 105055527
 * Last modified by: cadm_kafkama00
 * Created: Mon Sep 05 18:14:57 2016
 * Last modified: Tue Nov 26 15:54:38 2024
 * Model Version: 2.02
 * Description: Detection Algorithm for grid connection.

   HISTORY:
   V1.00  24.07.2020 Keller   created
   V1.01  07.08.2020 Huber  included function block from simulation
   V1.02  29.04.2021 Denk   VectorShift and LVRT function added
   V1.03  31.01.2022 Keller  add input for GCB_On

   V2.00  10.08.2023 Walch  Revision of parametrization, sensitivity and FRT selectivity
   V2.01  22.11.2023 Walch  Include grid observer
   10.01.2024 Walch  Include TP LVRT hold time for weak LVRT blocking
   V2.02  25.11.2024 Walch  Update grid observer for SS mains parallel vs. island plausibility check
 * modified Comment:
 ********************************************************************
 * Header for program GridStat
 ********************************************************************
 * Generated with B&R Automation Studio Target for Simulink V6.7.1
 * (ERT based)
 ********************************************************************/

#ifndef RTW_HEADER_GridStat_private_h_
#define RTW_HEADER_GridStat_private_h_
#include "rtwtypes.h"
#include "zero_crossing_types.h"
#include "GridStat.h"
#include <bur/plctypes.h>
#ifndef MIN
#define MIN(a,b)                       ((a) < (b) ? (a) : (b))
#endif

#ifndef MAX
#define MAX(a,b)                       ((a) > (b) ? (a) : (b))
#endif

#ifndef AST_ROUND
#define AST_ROUND(x)                   ((x)>=0?(long long)((x)+0.5):(long long)((x)-0.5))
#endif

extern int32_T div_nde_s32_floor(int32_T numerator, int32_T denominator, struct fGridStat* inst);
extern void GridStat_TofLvrtWeakBlk1_Init(rtDW_TofLvrtWeakBlk1_GridStat *localDW, struct fGridStat* inst);
extern void GridStat_TofLvrtWeakBlk1(plcbit rtu_IN, real32_T rtu_PT,
  rtB_TofLvrtWeakBlk1_GridStat *localB, rtDW_TofLvrtWeakBlk1_GridStat *localDW, struct fGridStat* inst);
extern void GridS_TpDetNabsProtTrigger_Init(rtDW_TpDetNabsProtTrigger_GridS
  *localDW, struct fGridStat* inst);
extern void GridStat_TpDetNabsProtTrigger(plcbit rtu_IN, real32_T rtu_PT,
  rtB_TpDetNabsProtTrigger_GridSt *localB, rtDW_TpDetNabsProtTrigger_GridS
  *localDW, struct fGridStat* inst);

#endif                                 /* RTW_HEADER_GridStat_private_h_ */
```

#### GridStat_types.h
```c
/********************************************************************
 * COPYRIGHT -- B&R Industrial Automation GmbH
 ********************************************************************
 * Program: GridStat
 * File: GridStat_types.h
 * Author: 105055527
 * Last modified by: cadm_kafkama00
 * Created: Mon Sep 05 18:14:57 2016
 * Last modified: Tue Nov 26 15:54:38 2024
 * Model Version: 2.02
 * Description: Detection Algorithm for grid connection.

   HISTORY:
   V1.00  24.07.2020 Keller   created
   V1.01  07.08.2020 Huber  included function block from simulation
   V1.02  29.04.2021 Denk   VectorShift and LVRT function added
   V1.03  31.01.2022 Keller  add input for GCB_On

   V2.00  10.08.2023 Walch  Revision of parametrization, sensitivity and FRT selectivity
   V2.01  22.11.2023 Walch  Include grid observer
   10.01.2024 Walch  Include TP LVRT hold time for weak LVRT blocking
   V2.02  25.11.2024 Walch  Update grid observer for SS mains parallel vs. island plausibility check
 * modified Comment:
 ********************************************************************
 * Header for program GridStat
 ********************************************************************
 * Generated with B&R Automation Studio Target for Simulink V6.7.1
 * (ERT based)
 ********************************************************************/

#ifndef RTW_HEADER_GridStat_types_h_
#define RTW_HEADER_GridStat_types_h_
#include "rtwtypes.h"

/* Model Code Variants */
#ifndef MIN
#define MIN(a,b)                       ((a) < (b) ? (a) : (b))
#endif

#ifndef MAX
#define MAX(a,b)                       ((a) > (b) ? (a) : (b))
#endif

#ifndef AST_ROUND
#define AST_ROUND(x)                   ((x)>=0?(long long)((x)+0.5):(long long)((x)-0.5))
#endif

/* Forward declaration for rtModel */

#endif                                 /* RTW_HEADER_GridStat_types_h_ */
```

#### fGridStat.c
```c
/********************************************************************
 * COPYRIGHT -- B&R Industrial Automation GmbH
 ********************************************************************
 * Program: GridStat
 * File: fGridStat.c
 * Author: 105055527
 * Last modified by: cadm_kafkama00
 * Created: Mon Sep 05 18:14:57 2016
 * Last modified: Tue Nov 26 15:54:38 2024
 * Model Version: 2.02
 * Description: Detection Algorithm for grid connection.

   HISTORY:
   V1.00  24.07.2020 Keller   created
   V1.01  07.08.2020 Huber  included function block from simulation
   V1.02  29.04.2021 Denk   VectorShift and LVRT function added
   V1.03  31.01.2022 Keller  add input for GCB_On

   V2.00  10.08.2023 Walch  Revision of parametrization, sensitivity and FRT selectivity
   V2.01  22.11.2023 Walch  Include grid observer
   10.01.2024 Walch  Include TP LVRT hold time for weak LVRT blocking
   V2.02  25.11.2024 Walch  Update grid observer for SS mains parallel vs. island plausibility check
 * modified Comment:
 ********************************************************************
 * Implementation of program GridStat
 ********************************************************************
 * Generated with B&R Automation Studio Target for Simulink V6.7.1
 * (ERT based)
 ********************************************************************/

#include <bur/plctypes.h>
#include "GridStat.h"
#include "rtwtypes.h"

/* Defines */
#define SS_TERMINATE 4
#define SS_OUTPUT 3
#define SS_INITIALIZE 2

/*  Data Types */

/**************************** GLOBAL DATA *************************************/
/*  Definitions */

/*  Declarations  */

/***************************** FILE SCOPE DATA ********************************/

/*************************** FUNCTIONS ****************************************/
#ifdef __cplusplus

unsigned long bur_heap_size = 6553500;

#endif

/*LEGACYMODE_VARIABLES*/
void fGridStat(struct fGridStat* inst)
{
  tag_RTM_GridStat* const GridStat_M = &(inst)->bur_GridStat;
	inst->bur_GridStat.blockIO = &(inst)->bur_BlockIO_GridStat;
	inst->bur_GridStat.prevZCSigState = &(inst)->bur_PrevZCSigStates_GridStat;
	inst->bur_GridStat.outputs = &(inst)->bur_ExternalOutputs_GridStat;
	inst->bur_GridStat.dwork = &(inst)->bur_D_Work_GridStat;

  switch (inst->ssMethodType)
  {
   case SS_INITIALIZE:
    /* call model initialize function */
    GridStat_initialize(GridStat_M, inst);
    break;

   case SS_OUTPUT:
    /* call model step function */
    GridStat_step(GridStat_M, inst);

    break;

   case SS_TERMINATE:
    /* call model terminate function */
    GridStat_terminate(GridStat_M, inst);
    break;
  }
}

/*****************************************************************************
   Function block sample time: 0.01s
 *****************************************************************************/

/*****************************************************************************
   B&R Automation Studio Target for Simulink Version: A6.7.1 (02-Dec-2022)
 *****************************************************************************/

/*======================== TOOL VERSION INFORMATION ==========================*
 * MATLAB 9.11 (R2021b)14-May-2021                                            *
 * Simulink 10.4 (R2021b)14-May-2021                                          *
 * Simulink Coder 9.6 (R2021b)14-May-2021                                     *
 * Embedded Coder 7.7 (R2021b)14-May-2021                                     *
 * Stateflow 10.5 (R2021b)14-May-2021                                         *
 *============================================================================*/

/*======================= LICENSE IN USE INFORMATION =========================*
 * matlab                                                                     *
 * matlab_coder                                                               *
 * real-time_workshop                                                         *
 * rtw_embedded_coder                                                         *
 * simulink                                                                   *
 *============================================================================*/
```

#### lGridStat.fun
```iecst
FUNCTION_BLOCK fGridStat
  VAR_INPUT
    ssMethodType: SINT;
  END_VAR
  VAR_INPUT
        Para : GridStatusDetection_PARA_Bus; (**)
  END_VAR
  VAR_INPUT
        In : GridStatusDetection_IN_Bus; (**)
  END_VAR
  VAR_OUTPUT
        Out : GridStatusDetection_OUT_Bus; (**)
  END_VAR
  VAR_OUTPUT
        Dbg : GridStatusDetection_DBG_Bus; (**)
  END_VAR
  VAR_INPUT
        Perm : GridStatusDetection_PERM_Bus; (**)
  END_VAR
  VAR_OUTPUT
        Version : UDINT := 0; (**)
  END_VAR
	VAR
		bur_BlockIO_GridStat : BlockIO_GridStat;
	END_VAR
	VAR
		bur_PrevZCSigStates_GridStat : PrevZCSigStates_GridStat;
	END_VAR
	VAR
		bur_ExternalOutputs_GridStat : ExternalOutputs_GridStat;
	END_VAR
	VAR
		bur_D_Work_GridStat : D_Work_GridStat;
	END_VAR
	VAR
		bur_GridStat : tag_RTM_GridStat;
	END_VAR
END_FUNCTION_BLOCK
```

#### lGridStat.typ
```iecst
TYPE
	GridStatusDetection_DBG_Bus :  STRUCT
		rProt_norm :  REAL; (*rotational power normalized [-]*)
		bDetSpeedRise :  BOOL; (*trigger for grid loss detection based on rotational power or absolute speed threshold*)
		bDetIslandVPN :  BOOL; (*trigger for grid loss detection based on VPN (voltage, power, speed - Lukas Undevall)*)
		trigger_Nabs :  BOOL; (*trigger for grid loss detection - absolute speed threshold*)
		trigger_Prot :  BOOL; (*trigger for grid loss detection - rotational power*)
		trigger_PU :  BOOL; (*trigger for grid loss detection - power AND voltage (VPN)*)
		trigger_N :  BOOL; (*trigger for grid loss detection - speed (VPN)*)
		trigger_U :  BOOL; (*trigger for grid loss detection - voltage (VPN)*)
		trigger_P :  BOOL; (*trigger for grid loss detection - power (VPN)*)
		trigger_VS :  BOOL; (*trigger for grid loss detection - VectorShift (VPN)*)
		block_LVRT_VPN :  BOOL; (*trigger for grid loss detection - LVRT (VPN) block bit for detection*)
		trigger_LVRT_NoDelay :  BOOL; (*trigger for grid loss detection - VectorShift (VPN)*)
		rCorrFac_rN_set_Norm :  REAL; (*correction factor for engine speed reference (rpm)*)
		block_LVRT_speedAbs :  BOOL; (*trigger for grid loss detection - LVRT (speedAbs/rot.pow.) block bit for detection*)
		bDetGridObserver :  BOOL; (*trigger for grid loss detection based on Grid Observer*)
		ru_obs :  ARRAY[0..8] OF REAL; (*Std Grid Observer input*)
		ru_obs_strong :  ARRAY[0..8] OF REAL; (*Strong Grid Observer input*)
		ru_obs3 :  ARRAY[0..8] OF REAL; (*3rd model Grid Observer input*)
		ry_obs :  ARRAY[0..1] OF REAL; (*Grid Observer output*)
		rx_obs :  ARRAY[0..4] OF REAL; (*Std Grid Observer state*)
		rx_obs_strong :  ARRAY[0..4] OF REAL; (*Strong Grid Observer state*)
		rx_obs3 :  ARRAY[0..4] OF REAL; (*3rd model Grid Observer state*)
		rcorr :  ARRAY[0..4] OF REAL; (*Std Grid Observer correction*)
		rcorr_strong :  ARRAY[0..4] OF REAL; (*Strong Grid Observer correction*)
		rcorr3 :  ARRAY[0..4] OF REAL; (*3rd model Grid Observer correction*)
	END_STRUCT;

	GridStatusDetection_IN_Bus :  STRUCT
		rN_engAct :  REAL; (*engine speed (rpm)*)
		rU_norm :  REAL; (*normalized voltage ([p.u.])*)
		rP_norm :  REAL; (*normalized power ([p.u.])*)
		rQ_norm :  REAL; (*normalized reactive power ([p.u.])*)
		rUexc_norm :  REAL; (*normalized excitation voltage ([p.u.])*)
		rF_norm :  REAL; (*normalized frequency ([p.u.])*)
		rp2s_norm :  REAL; (*normalized boost pressure ([p.u.])*)
		rN_F_Offset_Norm :  REAL; (*engine speed setpoint offset (-)*)
		bMCB_On :  BOOL; (*mains circuit breaker feedback (-)*)
		bGCB_On :  BOOL; (*generator circuit breaker feedback (-)*)
		bReset :  BOOL; (*Reset filter (-)*)
		bVectorShift :  BOOL; (*VectorShift protection relays hardware output  (-)*)
		bLVRT :  BOOL; (*LVRT signal (-)*)
	END_STRUCT;

	GridStatusDetection_OUT_Bus :  STRUCT
		rN_F_Offset_Norm_corr :  REAL; (*engine speed setpoint offset, corrected for transition grid parallel to island (-)*)
		bGridStatus :  BOOL; (*Grid Status bit: True if grid-parallel operation detected, false otherwise (-)*)
	END_STRUCT;

	GridStatusDetection_PARA_Bus :  STRUCT
		bEnable :  BOOL; (*Enable the grid status detection function (-)*)
		rTi_Filt_speed :  REAL; (*filter time constant speed filter for calculation rotational power (s)*)
		rTi_Filt_factorNoffsetCorr :  REAL; (*filter time constant filter for correction factor of speed ref. offset (s)*)
		rTi_Tof_MCBfb :  REAL; (*Pulse time TOF for bMCB_fb (s)*)
		rProt_Norm_limit :  REAL; (*limit  normalized rotational power for grid detection  (-)*)
		rTi_Tp_DetectActive :  REAL; (*Pulse time Tp for detection (s)*)
		rThrs_DeltaN_norm :  REAL; (*limit for speed signal deviation for grid detection (p.u.)*)
		rP_Nom :  REAL; (*nominal engine electrical power (kW)*)
		rN_Nom :  REAL; (*nominal engine speed  (rpm)*)
		rJ_Engine :  REAL; (*module inertia (kgm^2)*)
		iSamples_derivative_PU :  INT; (*time difference for evaluation of power / voltage change (default 20ms = 2) (n Samples)*)
		iSamples_Tp_detect_VPN :  INT; (*time slot for evalution of violation for power, voltage and speed threshold (default 50ms = 5) (n Samples)*)
		iSamples_derivative_N :  INT; (*time difference for evaluation of speed change (default 20ms = 2) (n Samples)*)
		rThrs_U_norm :  REAL; (*threshold for change of normalized voltage per second (1/s)*)
		rThrs_U_norm_FRTBlock :  REAL; (*threshold for change of normalized voltage per second, after weak FRT blocking was active (1/s)*)
		iSamples_Tof_U_norm_FRTBlock :  INT; (*time for voltage change threshold rThrs_U_norm_FRTBlock to be active after weak FRT blocking (default 1s = 100) (n Samples)*)
		rThrs_P_norm :  REAL; (*threshold for change of normalized power per second (1/s)*)
		rThrs_N_eng :  REAL; (*threshold for change of speed per second (rpm/s)*)
		rTi_sampleRate :  REAL; (*sample rate of algorithm (default 10ms = 0.01s) (s)*)
		iDetectMode :  INT; (*selector for detection Method: 1-speedAbs/rot.pow.; 2-VPN detection; 3-combined (-)*)
		rThrs_LVRT_norm :  REAL; (*voltage threshold to avoid falsely detected positive LVRTs (p.u.)*)
		iSamples_Tp_LVRT_hold :  INT; (*hold time for LVRT caused blocking (default 3000ms = 300) (n Samples)*)
		bLimitedTriggerTime :  BOOL; (*limit time slot for evalution of violation for power, voltage and speed threshold to iTi_detect_PandU (-)*)
		bWeakFRTBlocking :  BOOL; (*blocking of detection only if grid event bit AND voltage below rThrs_LVRT_norm (-)*)
		bWeakFRTBlocking_VPN :  BOOL; (*blocking of VPN detection only if grid event bit AND voltage below rThrs_LVRT_norm (possibility to block only for VPN) (-)*)
		bWeakFRTBlocking_speedAbs :  BOOL; (*blocking of speedAbs/rot.pow. detection only if grid event bit AND voltage below rThrs_LVRT_norm (possibility to block only for speedAbs/rot.pow.) (-)*)
		iSensitivity_WeakBlocking :  INT; (*Sensitivity weak blocking strategy (-)*)
		bN_BypassFRTBlocking :  BOOL; (*Bypass FRT blocking if absolute speed deviation above threshold (-)*)
		bN_BypassFRTBlocking_VPN :  BOOL; (*Bypass FRT blocking of VPN detection if absolute speed deviation above threshold (possibility to block only for VPN) (-)*)
		bN_BypassFRTBlocking_speedAbs :  BOOL; (*Bypass FRT blocking of speedAbs/rot.pow. detection if absolute speed deviation above threshold (possibility to block only for speedAbs/rot.pow.) (-)*)
		bEnable_SmoothDetection :  BOOL; (*Enable grid observer algorithm for detection of smooth islanding events (-)*)
		iSensitivity_SmoothDetection :  INT; (*Sensitivity of grid observer algorithm for detection of smooth islanding events (-)*)
	END_STRUCT;

	GridStatusDetection_PERM_Bus :  STRUCT
		dummy :  REAL; (**)
	END_STRUCT;

END_TYPE

TYPE
rtB_TofLvrtWeakBlk1_GridStat : STRUCT
	LogicalOperator1 : BOOL;
END_STRUCT;
rtDW_TofLvrtWeakBlk1_GridStat : STRUCT
	DiscreteTimeIntegrator_DSTATE : REAL;
	DiscreteTimeIntegrator_PrevRese : SINT;
	DiscreteTimeIntegrator_IC_LOADI : USINT;
END_STRUCT;
rtB_TpDetNabsProtTrigger_GridSt : STRUCT
	Merge : REAL;
	LogicalOperator1 : BOOL;
END_STRUCT;
rtDW_TpDetNabsProtTrigger_GridS : STRUCT
	DelayInput2_DSTATE : REAL;
	UnitDelay2_DSTATE : BOOL;
END_STRUCT;
BlockIO_GridStat : STRUCT
	BusConversion_InsertedFor_BusOu : GridStatusDetection_DBG_Bus;
	BusInput : GridStatusDetection_PARA_Bus;
	BusInput2 : GridStatusDetection_IN_Bus;
	BusInput1 : GridStatusDetection_PERM_Bus;
	UnitDelay : UDINT;
	TpUTrigger : rtB_TpDetNabsProtTrigger_GridSt;
	TpPTrigger : rtB_TpDetNabsProtTrigger_GridSt;
	TpNTrigger : rtB_TpDetNabsProtTrigger_GridSt;
	TpLvrtTrigHold2 : rtB_TpDetNabsProtTrigger_GridSt;
	TpLvrtBlockHold2 : rtB_TpDetNabsProtTrigger_GridSt;
	TpDetVPNTrigger : rtB_TpDetNabsProtTrigger_GridSt;
	TofLvrtWeakBlk2 : rtB_TofLvrtWeakBlk1_GridStat;
	TofAfterFRT : rtB_TofLvrtWeakBlk1_GridStat;
	TP_PU_trigger : rtB_TpDetNabsProtTrigger_GridSt;
	TofReset : rtB_TofLvrtWeakBlk1_GridStat;
	TofMcbFb : rtB_TofLvrtWeakBlk1_GridStat;
	TpProtTrigger : rtB_TpDetNabsProtTrigger_GridSt;
	TpNabsTrigger : rtB_TpDetNabsProtTrigger_GridSt;
	TpLvrtTrigHold1 : rtB_TpDetNabsProtTrigger_GridSt;
	TpLvrtBlockHold1 : rtB_TpDetNabsProtTrigger_GridSt;
	TpDetNabsProtTrigger : rtB_TpDetNabsProtTrigger_GridSt;
	TofLvrtWeakBlk1 : rtB_TofLvrtWeakBlk1_GridStat;
END_STRUCT;
D_Work_GridStat : STRUCT
	DiscreteTimeIntegrator_DSTATE : LREAL;
	TappedDelay_X : ARRAY[0..9] OF REAL;
	TappedDelay1_X : ARRAY[0..9] OF REAL;
	TappedDelay2_X : ARRAY[0..9] OF REAL;
	TappedDelay_X_l : ARRAY[0..9] OF REAL;
	TappedDelay2_X_b : ARRAY[0..9] OF REAL;
	TappedDelay3_X : ARRAY[0..9] OF REAL;
	TappedDelay5_X : ARRAY[0..9] OF REAL;
	TappedDelay4_X : ARRAY[0..9] OF REAL;
	TappedDelay1_X_m : ARRAY[0..9] OF REAL;
	DiscreteTimeIntegrator_DSTATE_j : REAL;
	UnitDelay_DSTATE : UDINT;
	U_past : ARRAY[0..999] OF REAL;
	err_past : ARRAY[0..999] OF REAL;
	err_min : REAL;
	err_act : REAL;
	err_max : REAL;
	err_act_temp : ARRAY[0..4] OF REAL;
	err_past_Q : ARRAY[0..999] OF REAL;
	err_min_Q : REAL;
	err_act_Q : REAL;
	err_max_Q : REAL;
	err_act_temp_Q : ARRAY[0..4] OF REAL;
	ctr_U : INT;
	ctr_err : INT;
	ctr_acterr : INT;
	ctr_release : INT;
	ctr_err_Q : INT;
	ctr_acterr_Q : INT;
	ctr_release_Q : INT;
	IslandDetected_DSTATE : BOOL;
	DiscreteTimeIntegrator_PrevRese : SINT;
	DiscreteTimeIntegrator_PrevRe_g : SINT;
	DiscreteTimeIntegrator_IC_LOADI : USINT;
	icLoad : BOOL;
	U_past_not_empty : BOOL;
	err_past_not_empty : BOOL;
	flag_window : BOOL;
	err_past_Q_not_empty : BOOL;
	flag_window_Q : BOOL;
	TpUTrigger : rtDW_TpDetNabsProtTrigger_GridS;
	TpPTrigger : rtDW_TpDetNabsProtTrigger_GridS;
	TpNTrigger : rtDW_TpDetNabsProtTrigger_GridS;
	TpLvrtTrigHold2 : rtDW_TpDetNabsProtTrigger_GridS;
	TpLvrtBlockHold2 : rtDW_TpDetNabsProtTrigger_GridS;
	TpDetVPNTrigger : rtDW_TpDetNabsProtTrigger_GridS;
	TofLvrtWeakBlk2 : rtDW_TofLvrtWeakBlk1_GridStat;
	TofAfterFRT : rtDW_TofLvrtWeakBlk1_GridStat;
	TP_PU_trigger : rtDW_TpDetNabsProtTrigger_GridS;
	TofReset : rtDW_TofLvrtWeakBlk1_GridStat;
	TofMcbFb : rtDW_TofLvrtWeakBlk1_GridStat;
	TpProtTrigger : rtDW_TpDetNabsProtTrigger_GridS;
	TpNabsTrigger : rtDW_TpDetNabsProtTrigger_GridS;
	TpLvrtTrigHold1 : rtDW_TpDetNabsProtTrigger_GridS;
	TpLvrtBlockHold1 : rtDW_TpDetNabsProtTrigger_GridS;
	TpDetNabsProtTrigger : rtDW_TpDetNabsProtTrigger_GridS;
	TofLvrtWeakBlk1 : rtDW_TofLvrtWeakBlk1_GridStat;
END_STRUCT;
PrevZCSigStates_GridStat : STRUCT
	IslandDetected_Reset_ZCE : USINT;
END_STRUCT;
ExternalOutputs_GridStat : STRUCT
	Out : GridStatusDetection_OUT_Bus;
	dbg : GridStatusDetection_DBG_Bus;
END_STRUCT;
tag_RTM_GridStat : STRUCT
	errorStatus : REFERENCE TO USINT;
	blockIO : REFERENCE TO BlockIO_GridStat;
	prevZCSigState : REFERENCE TO PrevZCSigStates_GridStat;
	outputs : REFERENCE TO ExternalOutputs_GridStat;
	dwork : REFERENCE TO D_Work_GridStat;
END_STRUCT;
RT_MODEL_GridStat : tag_RTM_GridStat;

END_TYPE
TYPE
END_TYPE
```

#### lib_properties.txt
```
For manual assignment to hardware configuration please
add the following additional include directories:

\Logical\MATLAB_includes\R2021b\

And the following additional build options:

-lm -D MODEL=GridStat -D NUMST=1 -D NCSTATES=0 -D HAVESTDIO -D MODEL_HAS_DYNAMICALLY_LOADED_SFCNS=0 -D CLASSIC_INTERFACE=0 -D ALLOCATIONFCN=0 -D TID01EQ=0 -D TERMFCN=1 -D ONESTEPFCN=1 -D MAT_FILE=0 -D MULTI_INSTANCE_CODE=1 -D INTEGER_CODE=0 -D MT=0
```
